LIN {X 0,Y 261.164,Z 765.318,A -85,B 0,C 180,E1 -18271.541,E2 -18271.541} C_VEL
LIN {X 0,Y 261.275,Z 764.733,A -85,B 0,C 180,E1 -18273.083,E2 -18273.083} C_VEL
LIN {X 0,Y 261.6,Z 762.413,A -85,B 0,C 180,E1 -18276.168,E2 -18276.168} C_VEL
LIN {X 0,Y 262.114,Z 759.545,A -85,B 0,C 180,E1 -18278.479,E2 -18278.479} C_VEL
LIN {X 0,Y 262.873,Z 755.654,A -85,B 0,C 180,E1 -18280.785,E2 -18280.785} C_VEL
LIN {X 0,Y 264.014,Z 750.637,A -85,B 0,C 180,E1 -18283.076,E2 -18283.076} C_VEL
LIN {X 0,Y 265.38,Z 744.319,A -85,B 0,C 180,E1 -18285.355,E2 -18285.355} C_VEL
LIN {X 0,Y 267.238,Z 736.403,A -85,B 0,C 180,E1 -18287.602,E2 -18287.602} C_VEL
LIN {X 0,Y 269.047,Z 728.334,A -85,B 0,C 180,E1 -18289.453,E2 -18289.453} C_VEL
LIN {X 0,Y 270.833,Z 718.491,A -85,B 0,C 180,E1 -18291.301,E2 -18291.301} C_VEL
LIN {X 0,Y 272.766,Z 707.41,A -85,B 0,C 180,E1 -18292.935,E2 -18292.935} C_VEL
LIN {X 0,Y 274.518,Z 696.535,A -85,B 0,C 180,E1 -18294.179,E2 -18294.179} C_VEL
LIN {X 0,Y 276.016,Z 684.51,A -85,B 0,C 180,E1 -18295.244,E2 -18295.244} C_VEL
LIN {X 0,Y 277.119,Z 672.156,A -85,B 0,C 180,E1 -18296.042,E2 -18296.042} C_VEL
LIN {X 0,Y 277.985,Z 659.336,A -85,B 0,C 180,E1 -18296.561,E2 -18296.561} C_VEL
LIN {X 0,Y 279.969,Z 592.257,A -85,B 0,C 180,E1 -18298.275,E2 -18298.275} C_VEL
LIN {X 0,Y 275.053,Z 579.197,A -85,B 0,C 180,E1 -18299.214,E2 -18299.214} C_VEL
LIN {X 0,Y 268.244,Z 564.095,A -85,B 0,C 180,E1 -18300.496,E2 -18300.496} C_VEL
LIN {X 0,Y 264.092,Z 555.532,A -85,B 0,C 180,E1 -18301.342,E2 -18301.342} C_VEL
LIN {X 0,Y 263.496,Z 553.165,A -85,B 0,C 180,E1 -18302.237,E2 -18302.237} C_VEL
LIN {X 0,Y 263.17,Z 551.724,A -85,B 0,C 180,E1 -18303.019,E2 -18303.019} C_VEL
LIN {X 0,Y 263.201,Z 551.693,A -85,B 0,C 180,E1 -18306.768,E2 -18306.768} C_VEL
LIN {X 0,Y 263.111,Z 551.696,A -85,B 0,C 180,E1 -18309.869,E2 -18309.869} C_VEL
LIN {X 0,Y 263.119,Z 551.693,A -85,B 0,C 180,E1 -18313.983,E2 -18313.983} C_VEL
LIN {X 0,Y 263.143,Z 551.706,A -85,B 0,C 180,E1 -18318.399,E2 -18318.399} C_VEL
LIN {X 0,Y 263.183,Z 551.673,A -85,B 0,C 180,E1 -18322.107,E2 -18322.107} C_VEL
LIN {X 0,Y 263.178,Z 551.702,A -85,B 0,C 180,E1 -18325.889,E2 -18325.889} C_VEL
LIN {X 0,Y 263.135,Z 551.7,A -85,B 0,C 180,E1 -18330.626,E2 -18330.626} C_VEL
LIN {X 0,Y 262.506,Z 551.779,A -85,B 0,C 180,E1 -18331.905,E2 -18331.905} C_VEL
LIN {X 0,Y 259.67,Z 552.137,A -85,B 0,C 180,E1 -18333.99,E2 -18333.99} C_VEL
LIN {X 0,Y 257.234,Z 552.441,A -85,B 0,C 180,E1 -18335.686,E2 -18335.686} C_VEL
LIN {X 0,Y 256.182,Z 552.564,A -85,B 0,C 180,E1 -18337.001,E2 -18337.001} C_VEL
LIN {X 0,Y 256.093,Z 552.571,A -85,B 0,C 180,E1 -18337.446,E2 -18337.446} C_VEL
LIN {X 0,Y 256.18,Z 552.572,A -85,B 0,C 180,E1 -18340.779,E2 -18340.779} C_VEL
LIN {X 0,Y 256.293,Z 552.544,A -85,B 0,C 180,E1 -18344.084,E2 -18344.084} C_VEL
LIN {X 0,Y 256.303,Z 552.548,A -85,B 0,C 180,E1 -18348.934,E2 -18348.934} C_VEL
LIN {X 0,Y 256.533,Z 552.526,A -85,B 0,C 180,E1 -18352.127,E2 -18352.127} C_VEL
LIN {X 0,Y 256.708,Z 552.501,A -85,B 0,C 180,E1 -18358.431,E2 -18358.431} C_VEL
LIN {X 0,Y 256.709,Z 552.503,A -85,B 0,C 180,E1 -18361.569,E2 -18361.569} C_VEL
LIN {X 0,Y 256.534,Z 552.526,A -85,B 0,C 180,E1 -18367.873,E2 -18367.873} C_VEL
LIN {X 0,Y 256.303,Z 552.545,A -85,B 0,C 180,E1 -18371.066,E2 -18371.066} C_VEL
LIN {X 0,Y 256.293,Z 552.545,A -85,B 0,C 180,E1 -18375.915,E2 -18375.915} C_VEL
LIN {X 0,Y 256.161,Z 552.568,A -85,B 0,C 180,E1 -18380.896,E2 -18380.896} C_VEL
LIN {X 0,Y 256.181,Z 552.573,A -85,B 0,C 180,E1 -18385.139,E2 -18385.139} C_VEL
LIN {X 0,Y 256.097,Z 552.584,A -85,B 0,C 180,E1 -18389.602,E2 -18389.602} C_VEL
LIN {X 0,Y 256.062,Z 552.59,A -85,B 0,C 180,E1 -18393.294,E2 -18393.294} C_VEL
LIN {X 0,Y 256.109,Z 552.557,A -85,B 0,C 180,E1 -18397.272,E2 -18397.272} C_VEL
LIN {X 0,Y 256.076,Z 552.575,A -85,B 0,C 180,E1 -18401.199,E2 -18401.199} C_VEL
LIN {X 0,Y 256.071,Z 552.585,A -85,B 0,C 180,E1 -18405.527,E2 -18405.527} C_VEL
LIN {X 0,Y 256.128,Z 552.582,A -85,B 0,C 180,E1 -18408.813,E2 -18408.813} C_VEL
LIN {X 0,Y 256.184,Z 552.737,A -85,B 0,C 180,E1 -18411.859,E2 -18411.859} C_VEL
LIN {X 0,Y 258.574,Z 562.726,A -85,B 0,C 180,E1 -18416.141,E2 -18416.141} C_VEL
LIN {X 0,Y 259.723,Z 567.866,A -85,B 0,C 180,E1 -18418.095,E2 -18418.095} C_VEL
LIN {X 0,Y 266.611,Z 583.7,A -85,B 0,C 180,E1 -18419.536,E2 -18419.536} C_VEL
LIN {X 0,Y 268.93,Z 589.726,A -85,B 0,C 180,E1 -18420.006,E2 -18420.006} C_VEL
LIN {X 0,Y 272.869,Z 615.019,A -85,B 0,C 180,E1 -18421.224,E2 -18421.224} C_VEL
LIN {X 0,Y 273.054,Z 619.058,A -85,B 0,C 180,E1 -18421.363,E2 -18421.363} C_VEL
LIN {X 0,Y 271.099,Z 676.352,A -85,B 0,C 180,E1 -18422.866,E2 -18422.866} C_VEL
LIN {X 0,Y 269.902,Z 690.247,A -85,B 0,C 180,E1 -18423.52,E2 -18423.52} C_VEL
LIN {X 0,Y 268.425,Z 702.691,A -85,B 0,C 180,E1 -18424.407,E2 -18424.407} C_VEL
LIN {X 0,Y 266.768,Z 713.801,A -85,B 0,C 180,E1 -18425.487,E2 -18425.487} C_VEL
LIN {X 0,Y 264.711,Z 725.369,A -85,B 0,C 180,E1 -18426.947,E2 -18426.947} C_VEL
LIN {X 0,Y 262.615,Z 735.787,A -85,B 0,C 180,E1 -18428.617,E2 -18428.617} C_VEL
LIN {X 0,Y 260.748,Z 744.664,A -85,B 0,C 180,E1 -18430.395,E2 -18430.395} C_VEL
LIN {X 0,Y 258.813,Z 753.554,A -85,B 0,C 180,E1 -18432.622,E2 -18432.622} C_VEL
LIN {X 0,Y 257.095,Z 760.984,A -85,B 0,C 180,E1 -18434.95,E2 -18434.95} C_VEL
LIN {X 0,Y 255.752,Z 766.951,A -85,B 0,C 180,E1 -18437.302,E2 -18437.302} C_VEL
LIN {X 0,Y 254.876,Z 771.673,A -85,B 0,C 180,E1 -18439.676,E2 -18439.676} C_VEL
LIN {X 0,Y 254.315,Z 775.286,A -85,B 0,C 180,E1 -18442.059,E2 -18442.059} C_VEL
LIN {X 0,Y 253.99,Z 778.347,A -85,B 0,C 180,E1 -18444.963,E2 -18444.963} C_VEL
LIN {X 0,Y 253.962,Z 779.544,A -85,B 0,C 180,E1 -18446.829,E2 -18446.829} C_VEL
LIN {X 0,Y 253.99,Z 780.152,A -85,B 0,C 180,E1 -18448.416,E2 -18448.416} C_VEL
LIN {X 0,Y 254.004,Z 780.51,A -85,B 0,C 180,E1 -18450.794,E2 -18450.794} C_VEL
LIN {X 0,Y 254.023,Z 782.645,A -85,B 0,C 180,E1 -18453.173,E2 -18453.173} C_VEL
LIN {X 0,Y 254.202,Z 783.607,A -85,B 0,C 180,E1 -18455.553,E2 -18455.553} C_VEL
LIN {X 0,Y 254.598,Z 783.41,A -85,B 0,C 180,E1 -18457.935,E2 -18457.935} C_VEL
LIN {X 0,Y 255.15,Z 782.591,A -85,B 0,C 180,E1 -18459.514,E2 -18459.514} C_VEL
LIN {X 0,Y 255.882,Z 781.29,A -85,B 0,C 180,E1 -18461.086,E2 -18461.086} C_VEL
LIN {X 0,Y 257.217,Z 778.306,A -85,B 0,C 180,E1 -18463.431,E2 -18463.431} C_VEL
LIN {X 0,Y 258.986,Z 774.096,A -85,B 0,C 180,E1 -18465.747,E2 -18465.747} C_VEL
LIN {X 0,Y 261.393,Z 768.401,A -85,B 0,C 180,E1 -18468.012,E2 -18468.012} C_VEL
LIN {X 0,Y 263.539,Z 762.327,A -85,B 0,C 180,E1 -18469.879,E2 -18469.879} C_VEL
LIN {X 0,Y 265.99,Z 754.985,A -85,B 0,C 180,E1 -18471.711,E2 -18471.711} C_VEL
LIN {X 0,Y 268.384,Z 746.866,A -85,B 0,C 180,E1 -18473.354,E2 -18473.354} C_VEL
LIN {X 0,Y 271.006,Z 736.903,A -85,B 0,C 180,E1 -18474.925,E2 -18474.925} C_VEL
LIN {X 0,Y 273.235,Z 727.291,A -85,B 0,C 180,E1 -18476.136,E2 -18476.136} C_VEL
LIN {X 0,Y 275.407,Z 716.047,A -85,B 0,C 180,E1 -18477.243,E2 -18477.243} C_VEL
LIN {X 0,Y 277.242,Z 703.03,A -85,B 0,C 180,E1 -18478.174,E2 -18478.174} C_VEL
LIN {X 0,Y 280.075,Z 679.812,A -85,B 0,C 180,E1 -18479.4,E2 -18479.4} C_VEL
LIN {X 0,Y 288.139,Z 623.235,A -85,B 0,C 180,E1 -18482.092,E2 -18482.092} C_VEL
LIN {X 0,Y 288.371,Z 616.794,A -85,B 0,C 180,E1 -18482.75,E2 -18482.75} C_VEL
LIN {X 0,Y 288.876,Z 615.038,A -85,B 0,C 180,E1 -18483.011,E2 -18483.011} C_VEL
LIN {X 0,Y 289.022,Z 612.57,A -85,B 0,C 180,E1 -18483.645,E2 -18483.645} C_VEL
LIN {X 0,Y 288.692,Z 608.855,A -85,B 0,C 180,E1 -18484.984,E2 -18484.984} C_VEL
LIN {X 0,Y 287.679,Z 606.935,A -85,B 0,C 180,E1 -18486.274,E2 -18486.274} C_VEL
LIN {X 0,Y 286.249,Z 605.014,A -85,B 0,C 180,E1 -18488.218,E2 -18488.218} C_VEL
LIN {X 0,Y 285.184,Z 603.787,A -85,B 0,C 180,E1 -18490.186,E2 -18490.186} C_VEL
LIN {X 0,Y 284.41,Z 603.27,A -85,B 0,C 180,E1 -18492.156,E2 -18492.156} C_VEL
LIN {X 0,Y 283.942,Z 603.412,A -85,B 0,C 180,E1 -18494.127,E2 -18494.127} C_VEL
LIN {X 0,Y 283.705,Z 604.229,A -85,B 0,C 180,E1 -18496.082,E2 -18496.082} C_VEL
LIN {X 0,Y 283.644,Z 606.871,A -85,B 0,C 180,E1 -18499.151,E2 -18499.151} C_VEL
LIN {X 0,Y 283.702,Z 608.841,A -85,B 0,C 180,E1 -18500.696,E2 -18500.696} C_VEL
LIN {X 0,Y 283.768,Z 613.689,A -85,B 0,C 180,E1 -18503.53,E2 -18503.53} C_VEL
LIN {X 0,Y 283.557,Z 617.891,A -85,B 0,C 180,E1 -18505.354,E2 -18505.354} C_VEL
LIN {X 0,Y 284.753,Z 629.469,A -85,B 0,C 180,E1 -18507.242,E2 -18507.242} C_VEL
LIN {X 0,Y 286.092,Z 642.547,A -85,B 0,C 180,E1 -18509.032,E2 -18509.032} C_VEL
LIN {X 0,Y 286.986,Z 654.978,A -85,B 0,C 180,E1 -18510.424,E2 -18510.424} C_VEL
LIN {X 0,Y 287.008,Z 657.879,A -85,B 0,C 180,E1 -18510.676,E2 -18510.676} C_VEL
LIN {X 0,Y 281.094,Z 703.082,A -85,B 0,C 180,E1 -18512.802,E2 -18512.802} C_VEL
LIN {X 0,Y 278.886,Z 715.353,A -85,B 0,C 180,E1 -18513.631,E2 -18513.631} C_VEL
LIN {X 0,Y 276.564,Z 725.576,A -85,B 0,C 180,E1 -18514.607,E2 -18514.607} C_VEL
LIN {X 0,Y 273.969,Z 735.191,A -85,B 0,C 180,E1 -18515.767,E2 -18515.767} C_VEL
LIN {X 0,Y 271.23,Z 744.198,A -85,B 0,C 180,E1 -18517.128,E2 -18517.128} C_VEL
LIN {X 0,Y 268.708,Z 751.51,A -85,B 0,C 180,E1 -18518.521,E2 -18518.521} C_VEL
LIN {X 0,Y 266.368,Z 757.638,A -85,B 0,C 180,E1 -18519.94,E2 -18519.94} C_VEL
LIN {X 0,Y 263.79,Z 763.91,A -85,B 0,C 180,E1 -18521.757,E2 -18521.757} C_VEL
LIN {X 0,Y 261.577,Z 769.036,A -85,B 0,C 180,E1 -18523.614,E2 -18523.614} C_VEL
LIN {X 0,Y 259.179,Z 773.831,A -85,B 0,C 180,E1 -18525.874,E2 -18525.874} C_VEL
LIN {X 0,Y 257.853,Z 776.163,A -85,B 0,C 180,E1 -18527.406,E2 -18527.406} C_VEL
LIN {X 0,Y 256.787,Z 777.941,A -85,B 0,C 180,E1 -18528.955,E2 -18528.955} C_VEL
LIN {X 0,Y 255.908,Z 779.221,A -85,B 0,C 180,E1 -18530.516,E2 -18530.516} C_VEL
LIN {X 0,Y 254.98,Z 780.156,A -85,B 0,C 180,E1 -18532.876,E2 -18532.876} C_VEL
LIN {X 0,Y 254.312,Z 779.949,A -85,B 0,C 180,E1 -18535.244,E2 -18535.244} C_VEL
LIN {X 0,Y 254.099,Z 779.107,A -85,B 0,C 180,E1 -18536.829,E2 -18536.829} C_VEL
LIN {X 0,Y 254.042,Z 777.756,A -85,B 0,C 180,E1 -18538.415,E2 -18538.415} C_VEL
LIN {X 0,Y 253.998,Z 774.661,A -85,B 0,C 180,E1 -18540.793,E2 -18540.793} C_VEL
LIN {X 0,Y 254.205,Z 770.236,A -85,B 0,C 180,E1 -18543.17,E2 -18543.17} C_VEL
LIN {X 0,Y 254.33,Z 765.193,A -85,B 0,C 180,E1 -18545.165,E2 -18545.165} C_VEL
LIN {X 0,Y 254.692,Z 758.914,A -85,B 0,C 180,E1 -18547.133,E2 -18547.133} C_VEL
LIN {X 0,Y 254.949,Z 752.669,A -85,B 0,C 180,E1 -18548.721,E2 -18548.721} C_VEL
LIN {X 0,Y 255.484,Z 744.165,A -85,B 0,C 180,E1 -18550.501,E2 -18550.501} C_VEL
LIN {X 0,Y 256.12,Z 734.618,A -85,B 0,C 180,E1 -18552.077,E2 -18552.077} C_VEL
LIN {X 0,Y 256.642,Z 725.68,A -85,B 0,C 180,E1 -18553.259,E2 -18553.259} C_VEL
LIN {X 0,Y 257.255,Z 714.434,A -85,B 0,C 180,E1 -18554.436,E2 -18554.436} C_VEL
LIN {X 0,Y 257.657,Z 702.446,A -85,B 0,C 180,E1 -18555.322,E2 -18555.322} C_VEL
LIN {X 0,Y 258.25,Z 687.986,A -85,B 0,C 180,E1 -18556.045,E2 -18556.045} C_VEL
LIN {X 0,Y 259.335,Z 642.712,A -85,B 0,C 180,E1 -18558.044,E2 -18558.044} C_VEL
LIN {X 0,Y 257.654,Z 620.795,A -85,B 0,C 180,E1 -18559.034,E2 -18559.034} C_VEL
LIN {X 0,Y 257.61,Z 617.12,A -85,B 0,C 180,E1 -18559.265,E2 -18559.265} C_VEL
LIN {X 0,Y 259.319,Z 596.268,A -85,B 0,C 180,E1 -18563.987,E2 -18563.987} C_VEL
LIN {X 0,Y 261.02,Z 578.045,A -85,B 0,C 180,E1 -18568.112,E2 -18568.112} C_VEL
LIN {X 0,Y 260.619,Z 574.104,A -85,B 0,C 180,E1 -18569.039,E2 -18569.039} C_VEL
LIN {X 0,Y 256.597,Z 554.39,A -85,B 0,C 180,E1 -18573.892,E2 -18573.892} C_VEL
LIN {X 0,Y 256.23,Z 552.679,A -85,B 0,C 180,E1 -18574.402,E2 -18574.402} C_VEL
LIN {X 0,Y 256.133,Z 552.582,A -85,B 0,C 180,E1 -18577.275,E2 -18577.275} C_VEL
LIN {X 0,Y 256.06,Z 552.532,A -85,B 0,C 180,E1 -18581.203,E2 -18581.203} C_VEL
LIN {X 0,Y 256.058,Z 552.579,A -85,B 0,C 180,E1 -18585.53,E2 -18585.53} C_VEL
LIN {X 0,Y 256.058,Z 552.558,A -85,B 0,C 180,E1 -18588.796,E2 -18588.796} C_VEL
LIN {X 0,Y 256.134,Z 552.57,A -85,B 0,C 180,E1 -18592.867,E2 -18592.867} C_VEL
LIN {X 0,Y 256.153,Z 552.695,A -85,B 0,C 180,E1 -18596.5,E2 -18596.5} C_VEL
LIN {X 0,Y 256.89,Z 555.635,A -85,B 0,C 180,E1 -18597.795,E2 -18597.795} C_VEL
LIN {X 0,Y 264.902,Z 572.152,A -85,B 0,C 180,E1 -18599.454,E2 -18599.454} C_VEL
LIN {X 0,Y 271.815,Z 588.544,A -85,B 0,C 180,E1 -18600.806,E2 -18600.806} C_VEL
LIN {X 0,Y 273.595,Z 593.413,A -85,B 0,C 180,E1 -18601.159,E2 -18601.159} C_VEL
LIN {X 0,Y 271.464,Z 661.742,A -85,B 0,C 180,E1 -18602.955,E2 -18602.955} C_VEL
LIN {X 0,Y 270.465,Z 675.096,A -85,B 0,C 180,E1 -18603.576,E2 -18603.576} C_VEL
LIN {X 0,Y 269.157,Z 687.837,A -85,B 0,C 180,E1 -18604.478,E2 -18604.478} C_VEL
LIN {X 0,Y 267.605,Z 699.142,A -85,B 0,C 180,E1 -18605.565,E2 -18605.565} C_VEL
LIN {X 0,Y 265.672,Z 710.779,A -85,B 0,C 180,E1 -18607.032,E2 -18607.032} C_VEL
LIN {X 0,Y 263.921,Z 719.999,A -85,B 0,C 180,E1 -18608.489,E2 -18608.489} C_VEL
LIN {X 0,Y 262.068,Z 729.758,A -85,B 0,C 180,E1 -18610.413,E2 -18610.413} C_VEL
LIN {X 0,Y 260.246,Z 737.623,A -85,B 0,C 180,E1 -18612.312,E2 -18612.312} C_VEL
LIN {X 0,Y 258.368,Z 745.306,A -85,B 0,C 180,E1 -18614.619,E2 -18614.619} C_VEL
LIN {X 0,Y 256.723,Z 752.357,A -85,B 0,C 180,E1 -18617.348,E2 -18617.348} C_VEL
LIN {X 0,Y 255.59,Z 757.052,A -85,B 0,C 180,E1 -18619.703,E2 -18619.703} C_VEL
LIN {X 0,Y 254.885,Z 760.637,A -85,B 0,C 180,E1 -18622.074,E2 -18622.074} C_VEL
LIN {X 0,Y 254.515,Z 762.598,A -85,B 0,C 180,E1 -18623.765,E2 -18623.765} C_VEL
LIN {X 0,Y 254.194,Z 764.873,A -85,B 0,C 180,E1 -18626.829,E2 -18626.829} C_VEL
LIN {X 0,Y 254.096,Z 765.484,A -85,B 0,C 180,E1 -18628.414,E2 -18628.414} C_VEL
LIN {X 0,Y 254.064,Z 765.714,A -85,B 0,C 180,E1 -18629.999,E2 -18629.999} C_VEL
LIN {X 0,Y 254.095,Z 765.522,A -85,B 0,C 180,E1 -18631.584,E2 -18631.584} C_VEL
LIN {X 0,Y 254.192,Z 764.937,A -85,B 0,C 180,E1 -18633.169,E2 -18633.169} C_VEL
LIN {X 0,Y 254.534,Z 762.617,A -85,B 0,C 180,E1 -18636.34,E2 -18636.34} C_VEL
LIN {X 0,Y 255.077,Z 759.749,A -85,B 0,C 180,E1 -18638.715,E2 -18638.715} C_VEL
LIN {X 0,Y 255.91,Z 755.858,A -85,B 0,C 180,E1 -18641.082,E2 -18641.082} C_VEL
LIN {X 0,Y 257.1,Z 750.84,A -85,B 0,C 180,E1 -18643.434,E2 -18643.434} C_VEL
LIN {X 0,Y 258.531,Z 744.522,A -85,B 0,C 180,E1 -18645.772,E2 -18645.772} C_VEL
LIN {X 0,Y 260.488,Z 736.605,A -85,B 0,C 180,E1 -18648.074,E2 -18648.074} C_VEL
LIN {X 0,Y 262.351,Z 728.536,A -85,B 0,C 180,E1 -18649.97,E2 -18649.97} C_VEL
LIN {X 0,Y 264.24,Z 718.692,A -85,B 0,C 180,E1 -18651.86,E2 -18651.86} C_VEL
LIN {X 0,Y 266.263,Z 707.609,A -85,B 0,C 180,E1 -18653.528,E2 -18653.528} C_VEL
LIN {X 0,Y 268.081,Z 696.733,A -85,B 0,C 180,E1 -18654.799,E2 -18654.799} C_VEL
LIN {X 0,Y 269.634,Z 684.707,A -85,B 0,C 180,E1 -18655.885,E2 -18655.885} C_VEL
LIN {X 0,Y 270.773,Z 672.349,A -85,B 0,C 180,E1 -18656.7,E2 -18656.7} C_VEL
LIN {X 0,Y 271.674,Z 659.519,A -85,B 0,C 180,E1 -18657.228,E2 -18657.228} C_VEL
LIN {X 0,Y 273.728,Z 593.61,A -85,B 0,C 180,E1 -18658.946,E2 -18658.946} C_VEL
LIN {X 0,Y 266.65,Z 575.931,A -85,B 0,C 180,E1 -18660.336,E2 -18660.336} C_VEL
LIN {X 0,Y 258.475,Z 558.972,A -85,B 0,C 180,E1 -18661.954,E2 -18661.954} C_VEL
LIN {X 0,Y 256.796,Z 555.428,A -85,B 0,C 180,E1 -18662.39,E2 -18662.39} C_VEL
LIN {X 0,Y 256.138,Z 552.622,A -85,B 0,C 180,E1 -18663.719,E2 -18663.719} C_VEL
LIN {X 0,Y 256.127,Z 552.578,A -85,B 0,C 180,E1 -18667.274,E2 -18667.274} C_VEL
LIN {X 0,Y 256.053,Z 552.584,A -85,B 0,C 180,E1 -18671.201,E2 -18671.201} C_VEL
LIN {X 0,Y 256.057,Z 552.569,A -85,B 0,C 180,E1 -18675.528,E2 -18675.528} C_VEL
LIN {X 0,Y 256.079,Z 552.582,A -85,B 0,C 180,E1 -18678.801,E2 -18678.801} C_VEL
LIN {X 0,Y 256.149,Z 552.557,A -85,B 0,C 180,E1 -18682.87,E2 -18682.87} C_VEL
LIN {X 0,Y 256.08,Z 552.582,A -85,B 0,C 180,E1 -18686.709,E2 -18686.709} C_VEL
LIN {X 0,Y 256.133,Z 552.572,A -85,B 0,C 180,E1 -18691.404,E2 -18691.404} C_VEL
LIN {X 0,Y 256.161,Z 552.574,A -85,B 0,C 180,E1 -18695.698,E2 -18695.698} C_VEL
LIN {X 0,Y 256.093,Z 552.571,A -85,B 0,C 180,E1 -18697.446,E2 -18697.446} C_VEL
LIN {X 0,Y 255.437,Z 552.656,A -85,B 0,C 180,E1 -18698.76,E2 -18698.76} C_VEL
LIN {X 0,Y 252.66,Z 553.011,A -85,B 0,C 180,E1 -18700.904,E2 -18700.904} C_VEL
LIN {X 0,Y 250.299,Z 553.296,A -85,B 0,C 180,E1 -18702.649,E2 -18702.649} C_VEL
LIN {X 0,Y 249.279,Z 553.417,A -85,B 0,C 180,E1 -18704,E2 -18704} C_VEL
LIN {X 0,Y 249.191,Z 553.428,A -85,B 0,C 180,E1 -18704.457,E2 -18704.457} C_VEL
LIN {X 0,Y 249.246,Z 553.43,A -85,B 0,C 180,E1 -18708.616,E2 -18708.616} C_VEL
LIN {X 0,Y 249.475,Z 553.401,A -85,B 0,C 180,E1 -18711.903,E2 -18711.903} C_VEL
LIN {X 0,Y 249.43,Z 553.396,A -85,B 0,C 180,E1 -18716.769,E2 -18716.769} C_VEL
LIN {X 0,Y 249.729,Z 553.378,A -85,B 0,C 180,E1 -18720,E2 -18720} C_VEL
LIN {X 0,Y 249.431,Z 553.398,A -85,B 0,C 180,E1 -18723.23,E2 -18723.23} C_VEL
LIN {X 0,Y 249.478,Z 553.404,A -85,B 0,C 180,E1 -18728.097,E2 -18728.097} C_VEL
LIN {X 0,Y 249.247,Z 553.426,A -85,B 0,C 180,E1 -18731.384,E2 -18731.384} C_VEL
LIN {X 0,Y 249.235,Z 553.424,A -85,B 0,C 180,E1 -18736.379,E2 -18736.379} C_VEL
LIN {X 0,Y 249.081,Z 553.447,A -85,B 0,C 180,E1 -18741.519,E2 -18741.519} C_VEL
LIN {X 0,Y 249.124,Z 553.448,A -85,B 0,C 180,E1 -18745.482,E2 -18745.482} C_VEL
LIN {X 0,Y 249.066,Z 553.461,A -85,B 0,C 180,E1 -18748.99,E2 -18748.99} C_VEL
LIN {X 0,Y 249.025,Z 553.465,A -85,B 0,C 180,E1 -18752.427,E2 -18752.427} C_VEL
LIN {X 0,Y 249.024,Z 553.436,A -85,B 0,C 180,E1 -18756.346,E2 -18756.346} C_VEL
LIN {X 0,Y 249.03,Z 553.464,A -85,B 0,C 180,E1 -18760.473,E2 -18760.473} C_VEL
LIN {X 0,Y 249.015,Z 553.468,A -85,B 0,C 180,E1 -18764.876,E2 -18764.876} C_VEL
LIN {X 0,Y 249.077,Z 553.446,A -85,B 0,C 180,E1 -18767.378,E2 -18767.378} C_VEL
LIN {X 0,Y 249.119,Z 553.651,A -85,B 0,C 180,E1 -18771.056,E2 -18771.056} C_VEL
LIN {X 0,Y 250.889,Z 560.889,A -85,B 0,C 180,E1 -18774.327,E2 -18774.327} C_VEL
LIN {X 0,Y 252.416,Z 567.595,A -85,B 0,C 180,E1 -18777.053,E2 -18777.053} C_VEL
LIN {X 0,Y 259.177,Z 582.558,A -85,B 0,C 180,E1 -18778.535,E2 -18778.535} C_VEL
LIN {X 0,Y 263.074,Z 592.539,A -85,B 0,C 180,E1 -18779.36,E2 -18779.36} C_VEL
LIN {X 0,Y 266.842,Z 617.494,A -85,B 0,C 180,E1 -18780.591,E2 -18780.591} C_VEL
LIN {X 0,Y 264.803,Z 676.161,A -85,B 0,C 180,E1 -18782.165,E2 -18782.165} C_VEL
LIN {X 0,Y 263.58,Z 690.052,A -85,B 0,C 180,E1 -18782.833,E2 -18782.833} C_VEL
LIN {X 0,Y 262.025,Z 702.492,A -85,B 0,C 180,E1 -18783.734,E2 -18783.734} C_VEL
LIN {X 0,Y 260.31,Z 713.601,A -85,B 0,C 180,E1 -18784.837,E2 -18784.837} C_VEL
LIN {X 0,Y 258.165,Z 725.167,A -85,B 0,C 180,E1 -18786.327,E2 -18786.327} C_VEL
LIN {X 0,Y 255.999,Z 735.585,A -85,B 0,C 180,E1 -18788.036,E2 -18788.036} C_VEL
LIN {X 0,Y 254.118,Z 744.109,A -85,B 0,C 180,E1 -18789.777,E2 -18789.777} C_VEL
LIN {X 0,Y 252.363,Z 752.158,A -85,B 0,C 180,E1 -18791.797,E2 -18791.797} C_VEL
LIN {X 0,Y 250.528,Z 759.66,A -85,B 0,C 180,E1 -18794.128,E2 -18794.128} C_VEL
LIN {X 0,Y 248.79,Z 766.747,A -85,B 0,C 180,E1 -18796.94,E2 -18796.94} C_VEL
LIN {X 0,Y 247.858,Z 771.468,A -85,B 0,C 180,E1 -18799.381,E2 -18799.381} C_VEL
LIN {X 0,Y 247.267,Z 775.082,A -85,B 0,C 180,E1 -18801.831,E2 -18801.831} C_VEL
LIN {X 0,Y 247.009,Z 776.944,A -85,B 0,C 180,E1 -18803.466,E2 -18803.466} C_VEL
LIN {X 0,Y 246.882,Z 778.341,A -85,B 0,C 180,E1 -18805.102,E2 -18805.102} C_VEL
LIN {X 0,Y 246.865,Z 779.339,A -85,B 0,C 180,E1 -18806.737,E2 -18806.737} C_VEL
LIN {X 0,Y 246.9,Z 779.948,A -85,B 0,C 180,E1 -18808.37,E2 -18808.37} C_VEL
LIN {X 0,Y 246.939,Z 780.108,A -85,B 0,C 180,E1 -18811.021,E2 -18811.021} C_VEL
LIN {X 0,Y 246.945,Z 782.262,A -85,B 0,C 180,E1 -18813.264,E2 -18813.264} C_VEL
LIN {X 0,Y 247.089,Z 783.383,A -85,B 0,C 180,E1 -18815.429,E2 -18815.429} C_VEL
LIN {X 0,Y 247.563,Z 783.464,A -85,B 0,C 180,E1 -18818.162,E2 -18818.162} C_VEL
LIN {X 0,Y 248.162,Z 782.873,A -85,B 0,C 180,E1 -18819.785,E2 -18819.785} C_VEL
LIN {X 0,Y 248.944,Z 781.787,A -85,B 0,C 180,E1 -18821.399,E2 -18821.399} C_VEL
LIN {X 0,Y 250.355,Z 779.09,A -85,B 0,C 180,E1 -18823.806,E2 -18823.806} C_VEL
LIN {X 0,Y 252.25,Z 775.164,A -85,B 0,C 180,E1 -18826.179,E2 -18826.179} C_VEL
LIN {X 0,Y 254.791,Z 769.872,A -85,B 0,C 180,E1 -18828.496,E2 -18828.496} C_VEL
LIN {X 0,Y 257.614,Z 763.042,A -85,B 0,C 180,E1 -18830.774,E2 -18830.774} C_VEL
LIN {X 0,Y 260.063,Z 756.333,A -85,B 0,C 180,E1 -18832.517,E2 -18832.517} C_VEL
LIN {X 0,Y 262.392,Z 749.327,A -85,B 0,C 180,E1 -18834.036,E2 -18834.036} C_VEL
LIN {X 0,Y 265.402,Z 739.699,A -85,B 0,C 180,E1 -18835.699,E2 -18835.699} C_VEL
LIN {X 0,Y 268.119,Z 729.217,A -85,B 0,C 180,E1 -18837.094,E2 -18837.094} C_VEL
LIN {X 0,Y 270.291,Z 719.596,A -85,B 0,C 180,E1 -18838.119,E2 -18838.119} C_VEL
LIN {X 0,Y 272.514,Z 707.097,A -85,B 0,C 180,E1 -18839.13,E2 -18839.13} C_VEL
LIN {X 0,Y 274.79,Z 689.707,A -85,B 0,C 180,E1 -18840.129,E2 -18840.129} C_VEL
LIN {X 0,Y 284.58,Z 625.063,A -85,B 0,C 180,E1 -18843.284,E2 -18843.284} C_VEL
LIN {X 0,Y 284.762,Z 618.517,A -85,B 0,C 180,E1 -18843.946,E2 -18843.946} C_VEL
LIN {X 0,Y 284.547,Z 616.843,A -85,B 0,C 180,E1 -18844.365,E2 -18844.365} C_VEL
LIN {X 0,Y 284.339,Z 614.215,A -85,B 0,C 180,E1 -18845.347,E2 -18845.347} C_VEL
LIN {X 0,Y 282.791,Z 611.68,A -85,B 0,C 180,E1 -18847.319,E2 -18847.319} C_VEL
LIN {X 0,Y 281.504,Z 610.085,A -85,B 0,C 180,E1 -18849.29,E2 -18849.29} C_VEL
LIN {X 0,Y 280.517,Z 609.207,A -85,B 0,C 180,E1 -18851.27,E2 -18851.27} C_VEL
LIN {X 0,Y 279.851,Z 609.01,A -85,B 0,C 180,E1 -18853.257,E2 -18853.257} C_VEL
LIN {X 0,Y 279.407,Z 609.494,A -85,B 0,C 180,E1 -18855.228,E2 -18855.228} C_VEL
LIN {X 0,Y 279.15,Z 610.667,A -85,B 0,C 180,E1 -18857.175,E2 -18857.175} C_VEL
LIN {X 0,Y 279.082,Z 613.325,A -85,B 0,C 180,E1 -18859.915,E2 -18859.915} C_VEL
LIN {X 0,Y 278.948,Z 617.866,A -85,B 0,C 180,E1 -18862.795,E2 -18862.795} C_VEL
LIN {X 0,Y 280.508,Z 623.055,A -85,B 0,C 180,E1 -18864.563,E2 -18864.563} C_VEL
LIN {X 0,Y 281.613,Z 636.846,A -85,B 0,C 180,E1 -18866.787,E2 -18866.787} C_VEL
LIN {X 0,Y 282.492,Z 649.442,A -85,B 0,C 180,E1 -18868.473,E2 -18868.473} C_VEL
LIN {X 0,Y 282.893,Z 659.147,A -85,B 0,C 180,E1 -18869.542,E2 -18869.542} C_VEL
LIN {X 0,Y 276.762,Z 702.685,A -85,B 0,C 180,E1 -18871.619,E2 -18871.619} C_VEL
LIN {X 0,Y 274.619,Z 713.885,A -85,B 0,C 180,E1 -18872.364,E2 -18872.364} C_VEL
LIN {X 0,Y 271.734,Z 725.886,A -85,B 0,C 180,E1 -18873.503,E2 -18873.503} C_VEL
LIN {X 0,Y 268.986,Z 735.508,A -85,B 0,C 180,E1 -18874.669,E2 -18874.669} C_VEL
LIN {X 0,Y 265.709,Z 745.328,A -85,B 0,C 180,E1 -18876.211,E2 -18876.211} C_VEL
LIN {X 0,Y 262.994,Z 752.402,A -85,B 0,C 180,E1 -18877.617,E2 -18877.617} C_VEL
LIN {X 0,Y 259.943,Z 759.741,A -85,B 0,C 180,E1 -18879.422,E2 -18879.422} C_VEL
LIN {X 0,Y 256.743,Z 766.755,A -85,B 0,C 180,E1 -18881.651,E2 -18881.651} C_VEL
LIN {X 0,Y 254.046,Z 771.968,A -85,B 0,C 180,E1 -18883.94,E2 -18883.94} C_VEL
LIN {X 0,Y 251.687,Z 775.909,A -85,B 0,C 180,E1 -18886.27,E2 -18886.27} C_VEL
LIN {X 0,Y 249.871,Z 778.588,A -85,B 0,C 180,E1 -18888.645,E2 -18888.645} C_VEL
LIN {X 0,Y 248.925,Z 779.623,A -85,B 0,C 180,E1 -18890.247,E2 -18890.247} C_VEL
LIN {X 0,Y 247.793,Z 780.343,A -85,B 0,C 180,E1 -18893.072,E2 -18893.072} C_VEL
LIN {X 0,Y 247.244,Z 779.845,A -85,B 0,C 180,E1 -18895.108,E2 -18895.108} C_VEL
LIN {X 0,Y 247.026,Z 778.84,A -85,B 0,C 180,E1 -18896.738,E2 -18896.738} C_VEL
LIN {X 0,Y 246.933,Z 776.379,A -85,B 0,C 180,E1 -18899.185,E2 -18899.185} C_VEL
LIN {X 0,Y 246.984,Z 772.505,A -85,B 0,C 180,E1 -18901.631,E2 -18901.631} C_VEL
LIN {X 0,Y 247.232,Z 767.192,A -85,B 0,C 180,E1 -18904.075,E2 -18904.075} C_VEL
LIN {X 0,Y 247.541,Z 760.096,A -85,B 0,C 180,E1 -18906.521,E2 -18906.521} C_VEL
LIN {X 0,Y 247.807,Z 754.111,A -85,B 0,C 180,E1 -18908.152,E2 -18908.152} C_VEL
LIN {X 0,Y 248.213,Z 746.906,A -85,B 0,C 180,E1 -18909.781,E2 -18909.781} C_VEL
LIN {X 0,Y 248.789,Z 738.186,A -85,B 0,C 180,E1 -18911.405,E2 -18911.405} C_VEL
LIN {X 0,Y 249.484,Z 727.082,A -85,B 0,C 180,E1 -18913.024,E2 -18913.024} C_VEL
LIN {X 0,Y 250.05,Z 717.155,A -85,B 0,C 180,E1 -18914.133,E2 -18914.133} C_VEL
LIN {X 0,Y 250.468,Z 705.188,A -85,B 0,C 180,E1 -18915.148,E2 -18915.148} C_VEL
LIN {X 0,Y 251.02,Z 691.705,A -85,B 0,C 180,E1 -18915.894,E2 -18915.894} C_VEL
LIN {X 0,Y 252.307,Z 643.671,A -85,B 0,C 180,E1 -18918.093,E2 -18918.093} C_VEL
LIN {X 0,Y 250.581,Z 620.824,A -85,B 0,C 180,E1 -18919.177,E2 -18919.177} C_VEL
LIN {X 0,Y 250.551,Z 617.295,A -85,B 0,C 180,E1 -18919.376,E2 -18919.376} C_VEL
LIN {X 0,Y 252.323,Z 596.175,A -85,B 0,C 180,E1 -18924.257,E2 -18924.257} C_VEL
LIN {X 0,Y 253.95,Z 579.679,A -85,B 0,C 180,E1 -18928.065,E2 -18928.065} C_VEL
LIN {X 0,Y 253.715,Z 575.774,A -85,B 0,C 180,E1 -18928.997,E2 -18928.997} C_VEL
LIN {X 0,Y 249.762,Z 556.397,A -85,B 0,C 180,E1 -18933.84,E2 -18933.84} C_VEL
LIN {X 0,Y 249.174,Z 553.587,A -85,B 0,C 180,E1 -18934.626,E2 -18934.626} C_VEL
LIN {X 0,Y 249.043,Z 553.458,A -85,B 0,C 180,E1 -18938.378,E2 -18938.378} C_VEL
LIN {X 0,Y 249.005,Z 553.406,A -85,B 0,C 180,E1 -18942.79,E2 -18942.79} C_VEL
LIN {X 0,Y 249.02,Z 553.462,A -85,B 0,C 180,E1 -18947.362,E2 -18947.362} C_VEL
LIN {X 0,Y 249.047,Z 553.437,A -85,B 0,C 180,E1 -18952.2,E2 -18952.2} C_VEL
LIN {X 0,Y 249.068,Z 553.518,A -85,B 0,C 180,E1 -18955.642,E2 -18955.642} C_VEL
LIN {X 0,Y 249.562,Z 555.442,A -85,B 0,C 180,E1 -18956.621,E2 -18956.621} C_VEL
LIN {X 0,Y 250.068,Z 556.886,A -85,B 0,C 180,E1 -18956.882,E2 -18956.882} C_VEL
LIN {X 0,Y 257.618,Z 571.872,A -85,B 0,C 180,E1 -18958.475,E2 -18958.475} C_VEL
LIN {X 0,Y 263.259,Z 584.586,A -85,B 0,C 180,E1 -18959.627,E2 -18959.627} C_VEL
LIN {X 0,Y 267.424,Z 595.311,A -85,B 0,C 180,E1 -18960.479,E2 -18960.479} C_VEL
LIN {X 0,Y 265.18,Z 661.963,A -85,B 0,C 180,E1 -18962.259,E2 -18962.259} C_VEL
LIN {X 0,Y 264.132,Z 675.31,A -85,B 0,C 180,E1 -18962.891,E2 -18962.891} C_VEL
LIN {X 0,Y 262.783,Z 688.049,A -85,B 0,C 180,E1 -18963.813,E2 -18963.813} C_VEL
LIN {X 0,Y 261.179,Z 699.352,A -85,B 0,C 180,E1 -18964.923,E2 -18964.923} C_VEL
LIN {X 0,Y 259.16,Z 710.988,A -85,B 0,C 180,E1 -18966.421,E2 -18966.421} C_VEL
LIN {X 0,Y 257.077,Z 721.435,A -85,B 0,C 180,E1 -18968.129,E2 -18968.129} C_VEL
LIN {X 0,Y 255.393,Z 729.966,A -85,B 0,C 180,E1 -18969.879,E2 -18969.879} C_VEL
LIN {X 0,Y 253.491,Z 737.83,A -85,B 0,C 180,E1 -18971.825,E2 -18971.825} C_VEL
LIN {X 0,Y 251.504,Z 745.513,A -85,B 0,C 180,E1 -18974.188,E2 -18974.188} C_VEL
LIN {X 0,Y 250.256,Z 750.756,A -85,B 0,C 180,E1 -18976.188,E2 -18976.188} C_VEL
LIN {X 0,Y 248.951,Z 755.843,A -85,B 0,C 180,E1 -18978.601,E2 -18978.601} C_VEL
LIN {X 0,Y 248.068,Z 759.785,A -85,B 0,C 180,E1 -18981.034,E2 -18981.034} C_VEL
LIN {X 0,Y 247.424,Z 763.002,A -85,B 0,C 180,E1 -18983.81,E2 -18983.81} C_VEL
LIN {X 0,Y 247.114,Z 765.078,A -85,B 0,C 180,E1 -18986.738,E2 -18986.738} C_VEL
LIN {X 0,Y 246.993,Z 765.918,A -85,B 0,C 180,E1 -18989.999,E2 -18989.999} C_VEL
LIN {X 0,Y 247.006,Z 765.726,A -85,B 0,C 180,E1 -18991.629,E2 -18991.629} C_VEL
LIN {X 0,Y 247.111,Z 765.141,A -85,B 0,C 180,E1 -18993.259,E2 -18993.259} C_VEL
LIN {X 0,Y 247.495,Z 762.821,A -85,B 0,C 180,E1 -18996.521,E2 -18996.521} C_VEL
LIN {X 0,Y 248.066,Z 759.953,A -85,B 0,C 180,E1 -18998.963,E2 -18998.963} C_VEL
LIN {X 0,Y 248.929,Z 756.062,A -85,B 0,C 180,E1 -19001.397,E2 -19001.397} C_VEL
LIN {X 0,Y 250.184,Z 751.044,A -85,B 0,C 180,E1 -19003.813,E2 -19003.813} C_VEL
LIN {X 0,Y 251.703,Z 744.724,A -85,B 0,C 180,E1 -19006.212,E2 -19006.212} C_VEL
LIN {X 0,Y 253.758,Z 736.807,A -85,B 0,C 180,E1 -19008.571,E2 -19008.571} C_VEL
LIN {X 0,Y 255.68,Z 728.738,A -85,B 0,C 180,E1 -19010.514,E2 -19010.514} C_VEL
LIN {X 0,Y 257.652,Z 718.894,A -85,B 0,C 180,E1 -19012.449,E2 -19012.449} C_VEL
LIN {X 0,Y 259.787,Z 707.809,A -85,B 0,C 180,E1 -19014.151,E2 -19014.151} C_VEL
LIN {X 0,Y 261.666,Z 696.931,A -85,B 0,C 180,E1 -19015.449,E2 -19015.449} C_VEL
LIN {X 0,Y 263.266,Z 684.904,A -85,B 0,C 180,E1 -19016.559,E2 -19016.559} C_VEL
LIN {X 0,Y 264.472,Z 672.541,A -85,B 0,C 180,E1 -19017.389,E2 -19017.389} C_VEL
LIN {X 0,Y 265.397,Z 659.703,A -85,B 0,C 180,E1 -19017.928,E2 -19017.928} C_VEL
LIN {X 0,Y 267.425,Z 595.25,A -85,B 0,C 180,E1 -19019.651,E2 -19019.651} C_VEL
LIN {X 0,Y 260.981,Z 579.13,A -85,B 0,C 180,E1 -19020.972,E2 -19020.972} C_VEL
LIN {X 0,Y 253.284,Z 563.062,A -85,B 0,C 180,E1 -19022.559,E2 -19022.559} C_VEL
LIN {X 0,Y 249.649,Z 555.829,A -85,B 0,C 180,E1 -19023.404,E2 -19023.404} C_VEL
LIN {X 0,Y 249.109,Z 553.695,A -85,B 0,C 180,E1 -19024.348,E2 -19024.348} C_VEL
LIN {X 0,Y 249.067,Z 553.451,A -85,B 0,C 180,E1 -19026.337,E2 -19026.337} C_VEL
LIN {X 0,Y 249.022,Z 553.452,A -85,B 0,C 180,E1 -19030.473,E2 -19030.473} C_VEL
LIN {X 0,Y 249.001,Z 553.446,A -85,B 0,C 180,E1 -19034.877,E2 -19034.877} C_VEL
LIN {X 0,Y 249.023,Z 553.464,A -85,B 0,C 180,E1 -19037.364,E2 -19037.364} C_VEL
LIN {X 0,Y 249.046,Z 553.431,A -85,B 0,C 180,E1 -19041.623,E2 -19041.623} C_VEL
LIN {X 0,Y 249.057,Z 553.463,A -85,B 0,C 180,E1 -19045.641,E2 -19045.641} C_VEL
LIN {X 0,Y 249.047,Z 553.463,A -85,B 0,C 180,E1 -19049.472,E2 -19049.472} C_VEL
LIN {X 0,Y 249.068,Z 553.449,A -85,B 0,C 180,E1 -19053.161,E2 -19053.161} C_VEL
LIN {X 0,Y 249.073,Z 553.451,A -85,B 0,C 180,E1 -19056.732,E2 -19056.732} C_VEL
LIN {X 0,Y 249.105,Z 553.454,A -85,B 0,C 180,E1 -19060.211,E2 -19060.211} C_VEL
LIN {X 0,Y 249.191,Z 553.428,A -85,B 0,C 180,E1 -19064.457,E2 -19064.457} C_VEL
LIN {X 0,Y 248.516,Z 553.524,A -85,B 0,C 180,E1 -19065.806,E2 -19065.806} C_VEL
LIN {X 0,Y 245.707,Z 553.874,A -85,B 0,C 180,E1 -19068.007,E2 -19068.007} C_VEL
LIN {X 0,Y 243.384,Z 554.153,A -85,B 0,C 180,E1 -19069.8,E2 -19069.8} C_VEL
LIN {X 0,Y 242.459,Z 554.268,A -85,B 0,C 180,E1 -19071.189,E2 -19071.189} C_VEL
LIN {X 0,Y 242.42,Z 554.277,A -85,B 0,C 180,E1 -19071.658,E2 -19071.658} C_VEL
LIN {X 0,Y 242.255,Z 554.303,A -85,B 0,C 180,E1 -19075.007,E2 -19075.007} C_VEL
LIN {X 0,Y 242.63,Z 554.252,A -85,B 0,C 180,E1 -19078.34,E2 -19078.34} C_VEL
LIN {X 0,Y 242.631,Z 554.256,A -85,B 0,C 180,E1 -19081.66,E2 -19081.66} C_VEL
LIN {X 0,Y 242.428,Z 554.286,A -85,B 0,C 180,E1 -19086.659,E2 -19086.659} C_VEL
LIN {X 0,Y 242.339,Z 554.28,A -85,B 0,C 180,E1 -19090.021,E2 -19090.021} C_VEL
LIN {X 0,Y 242.161,Z 554.31,A -85,B 0,C 180,E1 -19095.141,E2 -19095.141} C_VEL
LIN {X 0,Y 242.068,Z 554.331,A -85,B 0,C 180,E1 -19098.625,E2 -19098.625} C_VEL
LIN {X 0,Y 242.007,Z 554.328,A -85,B 0,C 180,E1 -19102.181,E2 -19102.181} C_VEL
LIN {X 0,Y 242.06,Z 554.324,A -85,B 0,C 180,E1 -19105.839,E2 -19105.839} C_VEL
LIN {X 0,Y 242.001,Z 554.339,A -85,B 0,C 180,E1 -19109.584,E2 -19109.584} C_VEL
LIN {X 0,Y 241.975,Z 554.344,A -85,B 0,C 180,E1 -19113.494,E2 -19113.494} C_VEL
LIN {X 0,Y 241.985,Z 554.317,A -85,B 0,C 180,E1 -19117.583,E2 -19117.583} C_VEL
LIN {X 0,Y 241.951,Z 554.328,A -85,B 0,C 180,E1 -19121.92,E2 -19121.92} C_VEL
LIN {X 0,Y 241.998,Z 554.328,A -85,B 0,C 180,E1 -19126.556,E2 -19126.556} C_VEL
LIN {X 0,Y 242.066,Z 554.398,A -85,B 0,C 180,E1 -19130.063,E2 -19130.063} C_VEL
LIN {X 0,Y 243.966,Z 562.14,A -85,B 0,C 180,E1 -19133.766,E2 -19133.766} C_VEL
LIN {X 0,Y 245.178,Z 567.218,A -85,B 0,C 180,E1 -19135.926,E2 -19135.926} C_VEL
LIN {X 0,Y 248.049,Z 573.648,A -85,B 0,C 180,E1 -19136.658,E2 -19136.658} C_VEL
LIN {X 0,Y 254.453,Z 587.836,A -85,B 0,C 180,E1 -19138.058,E2 -19138.058} C_VEL
LIN {X 0,Y 257.27,Z 595.421,A -85,B 0,C 180,E1 -19138.688,E2 -19138.688} C_VEL
LIN {X 0,Y 260.635,Z 618.502,A -85,B 0,C 180,E1 -19139.856,E2 -19139.856} C_VEL
LIN {X 0,Y 258.548,Z 675.97,A -85,B 0,C 180,E1 -19141.431,E2 -19141.431} C_VEL
LIN {X 0,Y 257.3,Z 689.856,A -85,B 0,C 180,E1 -19142.113,E2 -19142.113} C_VEL
LIN {X 0,Y 255.684,Z 702.294,A -85,B 0,C 180,E1 -19143.031,E2 -19143.031} C_VEL
LIN {X 0,Y 253.908,Z 713.401,A -85,B 0,C 180,E1 -19144.156,E2 -19144.156} C_VEL
LIN {X 0,Y 251.665,Z 724.966,A -85,B 0,C 180,E1 -19145.677,E2 -19145.677} C_VEL
LIN {X 0,Y 249.409,Z 735.383,A -85,B 0,C 180,E1 -19147.424,E2 -19147.424} C_VEL
LIN {X 0,Y 247.45,Z 743.906,A -85,B 0,C 180,E1 -19149.207,E2 -19149.207} C_VEL
LIN {X 0,Y 245.289,Z 753.148,A -85,B 0,C 180,E1 -19151.63,E2 -19151.63} C_VEL
LIN {X 0,Y 243.378,Z 760.577,A -85,B 0,C 180,E1 -19154.079,E2 -19154.079} C_VEL
LIN {X 0,Y 241.836,Z 766.542,A -85,B 0,C 180,E1 -19156.558,E2 -19156.558} C_VEL
LIN {X 0,Y 240.859,Z 771.264,A -85,B 0,C 180,E1 -19159.068,E2 -19159.068} C_VEL
LIN {X 0,Y 240.214,Z 774.877,A -85,B 0,C 180,E1 -19161.59,E2 -19161.59} C_VEL
LIN {X 0,Y 239.951,Z 776.74,A -85,B 0,C 180,E1 -19163.273,E2 -19163.273} C_VEL
LIN {X 0,Y 239.773,Z 778.339,A -85,B 0,C 180,E1 -19165.258,E2 -19165.258} C_VEL
LIN {X 0,Y 239.812,Z 779.744,A -85,B 0,C 180,E1 -19168.322,E2 -19168.322} C_VEL
LIN {X 0,Y 239.888,Z 779.875,A -85,B 0,C 180,E1 -19171.47,E2 -19171.47} C_VEL
LIN {X 0,Y 239.893,Z 781.754,A -85,B 0,C 180,E1 -19173.36,E2 -19173.36} C_VEL
LIN {X 0,Y 239.992,Z 782.984,A -85,B 0,C 180,E1 -19175.335,E2 -19175.335} C_VEL
LIN {X 0,Y 240.52,Z 783.518,A -85,B 0,C 180,E1 -19178.402,E2 -19178.402} C_VEL
LIN {X 0,Y 241.164,Z 783.128,A -85,B 0,C 180,E1 -19180.071,E2 -19180.071} C_VEL
LIN {X 0,Y 241.986,Z 782.154,A -85,B 0,C 180,E1 -19181.731,E2 -19181.731} C_VEL
LIN {X 0,Y 242.966,Z 780.691,A -85,B 0,C 180,E1 -19183.381,E2 -19183.381} C_VEL
LIN {X 0,Y 244.803,Z 777.564,A -85,B 0,C 180,E1 -19185.828,E2 -19185.828} C_VEL
LIN {X 0,Y 247.289,Z 773.197,A -85,B 0,C 180,E1 -19188.219,E2 -19188.219} C_VEL
LIN {X 0,Y 250.18,Z 767.252,A -85,B 0,C 180,E1 -19190.559,E2 -19190.559} C_VEL
LIN {X 0,Y 252.849,Z 761.15,A -85,B 0,C 180,E1 -19192.47,E2 -19192.47} C_VEL
LIN {X 0,Y 255.779,Z 753.729,A -85,B 0,C 180,E1 -19194.341,E2 -19194.341} C_VEL
LIN {X 0,Y 259.48,Z 743.381,A -85,B 0,C 180,E1 -19196.33,E2 -19196.33} C_VEL
LIN {X 0,Y 262.002,Z 735.351,A -85,B 0,C 180,E1 -19197.564,E2 -19197.564} C_VEL
LIN {X 0,Y 264.707,Z 725.401,A -85,B 0,C 180,E1 -19198.798,E2 -19198.798} C_VEL
LIN {X 0,Y 267.263,Z 714.077,A -85,B 0,C 180,E1 -19199.868,E2 -19199.868} C_VEL
LIN {X 0,Y 269.256,Z 702.524,A -85,B 0,C 180,E1 -19200.706,E2 -19200.706} C_VEL
LIN {X 0,Y 274.43,Z 668.532,A -85,B 0,C 180,E1 -19202.481,E2 -19202.481} C_VEL
LIN {X 0,Y 281.297,Z 626.742,A -85,B 0,C 180,E1 -19204.525,E2 -19204.525} C_VEL
LIN {X 0,Y 281.466,Z 622.311,A -85,B 0,C 180,E1 -19205.026,E2 -19205.026} C_VEL
LIN {X 0,Y 280.498,Z 619.783,A -85,B 0,C 180,E1 -19205.894,E2 -19205.894} C_VEL
LIN {X 0,Y 278.931,Z 617.731,A -85,B 0,C 180,E1 -19207.209,E2 -19207.209} C_VEL
LIN {X 0,Y 277.431,Z 615.891,A -85,B 0,C 180,E1 -19209.296,E2 -19209.296} C_VEL
LIN {X 0,Y 276.334,Z 614.937,A -85,B 0,C 180,E1 -19211.397,E2 -19211.397} C_VEL
LIN {X 0,Y 275.295,Z 614.922,A -85,B 0,C 180,E1 -19214.372,E2 -19214.372} C_VEL
LIN {X 0,Y 274.885,Z 615.785,A -85,B 0,C 180,E1 -19216.345,E2 -19216.345} C_VEL
LIN {X 0,Y 274.686,Z 618.134,A -85,B 0,C 180,E1 -19219.123,E2 -19219.123} C_VEL
LIN {X 0,Y 275.923,Z 622.423,A -85,B 0,C 180,E1 -19221.527,E2 -19221.527} C_VEL
LIN {X 0,Y 276.984,Z 625.736,A -85,B 0,C 180,E1 -19222.903,E2 -19222.903} C_VEL
LIN {X 0,Y 277.643,Z 628.423,A -85,B 0,C 180,E1 -19223.75,E2 -19223.75} C_VEL
LIN {X 0,Y 278.249,Z 641.035,A -85,B 0,C 180,E1 -19225.823,E2 -19225.823} C_VEL
LIN {X 0,Y 278.845,Z 653.763,A -85,B 0,C 180,E1 -19227.563,E2 -19227.563} C_VEL
LIN {X 0,Y 278.893,Z 661.315,A -85,B 0,C 180,E1 -19228.397,E2 -19228.397} C_VEL
LIN {X 0,Y 272.611,Z 702.728,A -85,B 0,C 180,E1 -19230.406,E2 -19230.406} C_VEL
LIN {X 0,Y 270.127,Z 714.863,A -85,B 0,C 180,E1 -19231.228,E2 -19231.228} C_VEL
LIN {X 0,Y 267.49,Z 725.131,A -85,B 0,C 180,E1 -19232.202,E2 -19232.202} C_VEL
LIN {X 0,Y 264.558,Z 734.74,A -85,B 0,C 180,E1 -19233.366,E2 -19233.366} C_VEL
LIN {X 0,Y 261.033,Z 744.672,A -85,B 0,C 180,E1 -19234.909,E2 -19234.909} C_VEL
LIN {X 0,Y 258.108,Z 751.893,A -85,B 0,C 180,E1 -19236.32,E2 -19236.32} C_VEL
LIN {X 0,Y 255.416,Z 757.941,A -85,B 0,C 180,E1 -19237.769,E2 -19237.769} C_VEL
LIN {X 0,Y 252.36,Z 764.151,A -85,B 0,C 180,E1 -19239.628,E2 -19239.628} C_VEL
LIN {X 0,Y 249.207,Z 770.133,A -85,B 0,C 180,E1 -19241.928,E2 -19241.928} C_VEL
LIN {X 0,Y 246.423,Z 774.571,A -85,B 0,C 180,E1 -19244.28,E2 -19244.28} C_VEL
LIN {X 0,Y 244.129,Z 777.648,A -85,B 0,C 180,E1 -19246.685,E2 -19246.685} C_VEL
LIN {X 0,Y 242.929,Z 779.1,A -85,B 0,C 180,E1 -19248.316,E2 -19248.316} C_VEL
LIN {X 0,Y 241.937,Z 780.028,A -85,B 0,C 180,E1 -19249.963,E2 -19249.963} C_VEL
LIN {X 0,Y 241.211,Z 780.363,A -85,B 0,C 180,E1 -19251.623,E2 -19251.623} C_VEL
LIN {X 0,Y 240.624,Z 780.211,A -85,B 0,C 180,E1 -19253.291,E2 -19253.291} C_VEL
LIN {X 0,Y 240.18,Z 779.588,A -85,B 0,C 180,E1 -19254.964,E2 -19254.964} C_VEL
LIN {X 0,Y 239.956,Z 778.468,A -85,B 0,C 180,E1 -19256.642,E2 -19256.642} C_VEL
LIN {X 0,Y 239.87,Z 775.656,A -85,B 0,C 180,E1 -19259.161,E2 -19259.161} C_VEL
LIN {X 0,Y 239.934,Z 771.56,A -85,B 0,C 180,E1 -19261.679,E2 -19261.679} C_VEL
LIN {X 0,Y 240.116,Z 768,A -85,B 0,C 180,E1 -19263.356,E2 -19263.356} C_VEL
LIN {X 0,Y 240.294,Z 762.714,A -85,B 0,C 180,E1 -19265.366,E2 -19265.366} C_VEL
LIN {X 0,Y 240.678,Z 755.492,A -85,B 0,C 180,E1 -19267.551,E2 -19267.551} C_VEL
LIN {X 0,Y 241.045,Z 748.523,A -85,B 0,C 180,E1 -19269.228,E2 -19269.228} C_VEL
LIN {X 0,Y 241.548,Z 740.057,A -85,B 0,C 180,E1 -19270.902,E2 -19270.902} C_VEL
LIN {X 0,Y 242.122,Z 731.023,A -85,B 0,C 180,E1 -19272.361,E2 -19272.361} C_VEL
LIN {X 0,Y 242.846,Z 719.452,A -85,B 0,C 180,E1 -19273.813,E2 -19273.813} C_VEL
LIN {X 0,Y 243.358,Z 708.405,A -85,B 0,C 180,E1 -19274.851,E2 -19274.851} C_VEL
LIN {X 0,Y 243.794,Z 694.903,A -85,B 0,C 180,E1 -19275.733,E2 -19275.733} C_VEL
LIN {X 0,Y 245.236,Z 644.331,A -85,B 0,C 180,E1 -19278.159,E2 -19278.159} C_VEL
LIN {X 0,Y 243.522,Z 621.09,A -85,B 0,C 180,E1 -19279.296,E2 -19279.296} C_VEL
LIN {X 0,Y 243.495,Z 617.23,A -85,B 0,C 180,E1 -19279.539,E2 -19279.539} C_VEL
LIN {X 0,Y 245.163,Z 597.85,A -85,B 0,C 180,E1 -19284.111,E2 -19284.111} C_VEL
LIN {X 0,Y 246.928,Z 579.712,A -85,B 0,C 180,E1 -19288.386,E2 -19288.386} C_VEL
LIN {X 0,Y 246.412,Z 575.299,A -85,B 0,C 180,E1 -19289.472,E2 -19289.472} C_VEL
LIN {X 0,Y 242.435,Z 555.922,A -85,B 0,C 180,E1 -19294.423,E2 -19294.423} C_VEL
LIN {X 0,Y 242.134,Z 554.445,A -85,B 0,C 180,E1 -19294.914,E2 -19294.914} C_VEL
LIN {X 0,Y 241.977,Z 554.308,A -85,B 0,C 180,E1 -19299.715,E2 -19299.715} C_VEL
LIN {X 0,Y 241.927,Z 554.303,A -85,B 0,C 180,E1 -19304.203,E2 -19304.203} C_VEL
LIN {X 0,Y 241.938,Z 554.327,A -85,B 0,C 180,E1 -19308.076,E2 -19308.076} C_VEL
LIN {X 0,Y 241.993,Z 554.319,A -85,B 0,C 180,E1 -19312.417,E2 -19312.417} C_VEL
LIN {X 0,Y 242.05,Z 554.502,A -85,B 0,C 180,E1 -19314.915,E2 -19314.915} C_VEL
LIN {X 0,Y 242.493,Z 556.177,A -85,B 0,C 180,E1 -19315.629,E2 -19315.629} C_VEL
LIN {X 0,Y 250.254,Z 571.289,A -85,B 0,C 180,E1 -19317.406,E2 -19317.406} C_VEL
LIN {X 0,Y 257.285,Z 586.85,A -85,B 0,C 180,E1 -19318.91,E2 -19318.91} C_VEL
LIN {X 0,Y 261.208,Z 596.939,A -85,B 0,C 180,E1 -19319.748,E2 -19319.748} C_VEL
LIN {X 0,Y 258.9,Z 662.781,A -85,B 0,C 180,E1 -19321.554,E2 -19321.554} C_VEL
LIN {X 0,Y 257.788,Z 676.351,A -85,B 0,C 180,E1 -19322.227,E2 -19322.227} C_VEL
LIN {X 0,Y 256.287,Z 689.349,A -85,B 0,C 180,E1 -19323.207,E2 -19323.207} C_VEL
LIN {X 0,Y 254.494,Z 701.144,A -85,B 0,C 180,E1 -19324.436,E2 -19324.436} C_VEL
LIN {X 0,Y 252.438,Z 712.484,A -85,B 0,C 180,E1 -19325.972,E2 -19325.972} C_VEL
LIN {X 0,Y 250.184,Z 723.103,A -85,B 0,C 180,E1 -19327.799,E2 -19327.799} C_VEL
LIN {X 0,Y 248.332,Z 731.863,A -85,B 0,C 180,E1 -19329.714,E2 -19329.714} C_VEL
LIN {X 0,Y 246.012,Z 740.772,A -85,B 0,C 180,E1 -19332.114,E2 -19332.114} C_VEL
LIN {X 0,Y 244.156,Z 747.937,A -85,B 0,C 180,E1 -19334.557,E2 -19334.557} C_VEL
LIN {X 0,Y 242.864,Z 752.77,A -85,B 0,C 180,E1 -19336.613,E2 -19336.613} C_VEL
LIN {X 0,Y 241.618,Z 757.464,A -85,B 0,C 180,E1 -19339.1,E2 -19339.1} C_VEL
LIN {X 0,Y 240.808,Z 761.049,A -85,B 0,C 180,E1 -19341.608,E2 -19341.608} C_VEL
LIN {X 0,Y 240.32,Z 763.43,A -85,B 0,C 180,E1 -19343.888,E2 -19343.888} C_VEL
LIN {X 0,Y 240.036,Z 765.283,A -85,B 0,C 180,E1 -19346.642,E2 -19346.642} C_VEL
LIN {X 0,Y 239.924,Z 766.122,A -85,B 0,C 180,E1 -19349.999,E2 -19349.999} C_VEL
LIN {X 0,Y 239.919,Z 765.93,A -85,B 0,C 180,E1 -19351.677,E2 -19351.677} C_VEL
LIN {X 0,Y 240.033,Z 765.345,A -85,B 0,C 180,E1 -19353.356,E2 -19353.356} C_VEL
LIN {X 0,Y 240.449,Z 763.025,A -85,B 0,C 180,E1 -19356.713,E2 -19356.713} C_VEL
LIN {X 0,Y 241.037,Z 760.157,A -85,B 0,C 180,E1 -19359.227,E2 -19359.227} C_VEL
LIN {X 0,Y 241.963,Z 756.265,A -85,B 0,C 180,E1 -19361.73,E2 -19361.73} C_VEL
LIN {X 0,Y 243.288,Z 751.247,A -85,B 0,C 180,E1 -19364.212,E2 -19364.212} C_VEL
LIN {X 0,Y 244.885,Z 744.927,A -85,B 0,C 180,E1 -19366.676,E2 -19366.676} C_VEL
LIN {X 0,Y 247.048,Z 737.009,A -85,B 0,C 180,E1 -19369.094,E2 -19369.094} C_VEL
LIN {X 0,Y 249.189,Z 728.144,A -85,B 0,C 180,E1 -19371.268,E2 -19371.268} C_VEL
LIN {X 0,Y 251.318,Z 717.997,A -85,B 0,C 180,E1 -19373.264,E2 -19373.264} C_VEL
LIN {X 0,Y 253.59,Z 706.587,A -85,B 0,C 180,E1 -19375,E2 -19375} C_VEL
LIN {X 0,Y 255.586,Z 695.366,A -85,B 0,C 180,E1 -19376.319,E2 -19376.319} C_VEL
LIN {X 0,Y 257.103,Z 683.964,A -85,B 0,C 180,E1 -19377.358,E2 -19377.358} C_VEL
LIN {X 0,Y 258.36,Z 670.914,A -85,B 0,C 180,E1 -19378.204,E2 -19378.204} C_VEL
LIN {X 0,Y 259.235,Z 658.384,A -85,B 0,C 180,E1 -19378.707,E2 -19378.707} C_VEL
LIN {X 0,Y 261.26,Z 597.047,A -85,B 0,C 180,E1 -19380.373,E2 -19380.373} C_VEL
LIN {X 0,Y 254.882,Z 581.211,A -85,B 0,C 180,E1 -19381.737,E2 -19381.737} C_VEL
LIN {X 0,Y 247.507,Z 565.943,A -85,B 0,C 180,E1 -19383.325,E2 -19383.325} C_VEL
LIN {X 0,Y 242.475,Z 556.117,A -85,B 0,C 180,E1 -19384.519,E2 -19384.519} C_VEL
LIN {X 0,Y 242.038,Z 554.426,A -85,B 0,C 180,E1 -19385.319,E2 -19385.319} C_VEL
LIN {X 0,Y 241.969,Z 554.329,A -85,B 0,C 180,E1 -19389.714,E2 -19389.714} C_VEL
LIN {X 0,Y 241.928,Z 554.329,A -85,B 0,C 180,E1 -19394.2,E2 -19394.2} C_VEL
LIN {X 0,Y 241.95,Z 554.347,A -85,B 0,C 180,E1 -19398.08,E2 -19398.08} C_VEL
LIN {X 0,Y 242.007,Z 554.311,A -85,B 0,C 180,E1 -19402.421,E2 -19402.421} C_VEL
LIN {X 0,Y 241.986,Z 554.339,A -85,B 0,C 180,E1 -19406.508,E2 -19406.508} C_VEL
LIN {X 0,Y 242.031,Z 554.336,A -85,B 0,C 180,E1 -19410.586,E2 -19410.586} C_VEL
LIN {X 0,Y 242.062,Z 554.332,A -85,B 0,C 180,E1 -19414.182,E2 -19414.182} C_VEL
LIN {X 0,Y 242.047,Z 554.32,A -85,B 0,C 180,E1 -19418.296,E2 -19418.296} C_VEL
LIN {X 0,Y 242.157,Z 554.305,A -85,B 0,C 180,E1 -19423.278,E2 -19423.278} C_VEL
LIN {X 0,Y 242.18,Z 554.312,A -85,B 0,C 180,E1 -19428.279,E2 -19428.279} C_VEL
LIN {X 0,Y 242.42,Z 554.277,A -85,B 0,C 180,E1 -19431.658,E2 -19431.658} C_VEL
LIN {X 0,Y 241.859,Z 554.359,A -85,B 0,C 180,E1 -19433.043,E2 -19433.043} C_VEL
LIN {X 0,Y 239.077,Z 554.701,A -85,B 0,C 180,E1 -19435.303,E2 -19435.303} C_VEL
LIN {X 0,Y 236.672,Z 554.993,A -85,B 0,C 180,E1 -19437.145,E2 -19437.145} C_VEL
LIN {X 0,Y 235.661,Z 555.122,A -85,B 0,C 180,E1 -19438.574,E2 -19438.574} C_VEL
LIN {X 0,Y 235.593,Z 555.129,A -85,B 0,C 180,E1 -19439.058,E2 -19439.058} C_VEL
LIN {X 0,Y 235.59,Z 555.132,A -85,B 0,C 180,E1 -19441.709,E2 -19441.709} C_VEL
LIN {X 0,Y 235.4,Z 555.162,A -85,B 0,C 180,E1 -19446.859,E2 -19446.859} C_VEL
LIN {X 0,Y 235.247,Z 555.164,A -85,B 0,C 180,E1 -19450.326,E2 -19450.326} C_VEL
LIN {X 0,Y 235.108,Z 555.184,A -85,B 0,C 180,E1 -19455.607,E2 -19455.607} C_VEL
LIN {X 0,Y 235.003,Z 555.213,A -85,B 0,C 180,E1 -19459.206,E2 -19459.206} C_VEL
LIN {X 0,Y 234.955,Z 555.212,A -85,B 0,C 180,E1 -19462.883,E2 -19462.883} C_VEL
LIN {X 0,Y 234.961,Z 555.205,A -85,B 0,C 180,E1 -19466.658,E2 -19466.658} C_VEL
LIN {X 0,Y 234.916,Z 555.216,A -85,B 0,C 180,E1 -19470.57,E2 -19470.57} C_VEL
LIN {X 0,Y 234.921,Z 555.208,A -85,B 0,C 180,E1 -19474.64,E2 -19474.64} C_VEL
LIN {X 0,Y 234.937,Z 555.215,A -85,B 0,C 180,E1 -19478.946,E2 -19478.946} C_VEL
LIN {X 0,Y 234.922,Z 555.206,A -85,B 0,C 180,E1 -19483.478,E2 -19483.478} C_VEL
LIN {X 0,Y 234.97,Z 555.203,A -85,B 0,C 180,E1 -19486.536,E2 -19486.536} C_VEL
LIN {X 0,Y 234.97,Z 555.249,A -85,B 0,C 180,E1 -19489.065,E2 -19489.065} C_VEL
LIN {X 0,Y 236.1,Z 559.501,A -85,B 0,C 180,E1 -19491.312,E2 -19491.312} C_VEL
LIN {X 0,Y 237.92,Z 567.072,A -85,B 0,C 180,E1 -19494.753,E2 -19494.753} C_VEL
LIN {X 0,Y 245.327,Z 582.799,A -85,B 0,C 180,E1 -19496.557,E2 -19496.557} C_VEL
LIN {X 0,Y 251.265,Z 597.038,A -85,B 0,C 180,E1 -19497.911,E2 -19497.911} C_VEL
LIN {X 0,Y 254.495,Z 619.574,A -85,B 0,C 180,E1 -19499.09,E2 -19499.09} C_VEL
LIN {X 0,Y 252.341,Z 675.779,A -85,B 0,C 180,E1 -19500.661,E2 -19500.661} C_VEL
LIN {X 0,Y 251.067,Z 689.661,A -85,B 0,C 180,E1 -19501.357,E2 -19501.357} C_VEL
LIN {X 0,Y 249.379,Z 702.095,A -85,B 0,C 180,E1 -19502.291,E2 -19502.291} C_VEL
LIN {X 0,Y 247.544,Z 713.201,A -85,B 0,C 180,E1 -19503.44,E2 -19503.44} C_VEL
LIN {X 0,Y 245.212,Z 724.765,A -85,B 0,C 180,E1 -19504.994,E2 -19504.994} C_VEL
LIN {X 0,Y 242.839,Z 735.181,A -85,B 0,C 180,E1 -19506.778,E2 -19506.778} C_VEL
LIN {X 0,Y 240.801,Z 743.704,A -85,B 0,C 180,E1 -19508.605,E2 -19508.605} C_VEL
LIN {X 0,Y 238.944,Z 751.457,A -85,B 0,C 180,E1 -19510.644,E2 -19510.644} C_VEL
LIN {X 0,Y 236.853,Z 759.253,A -85,B 0,C 180,E1 -19513.185,E2 -19513.185} C_VEL
LIN {X 0,Y 234.896,Z 766.338,A -85,B 0,C 180,E1 -19516.153,E2 -19516.153} C_VEL
LIN {X 0,Y 233.875,Z 771.06,A -85,B 0,C 180,E1 -19518.738,E2 -19518.738} C_VEL
LIN {X 0,Y 233.181,Z 774.673,A -85,B 0,C 180,E1 -19521.334,E2 -19521.334} C_VEL
LIN {X 0,Y 232.889,Z 776.536,A -85,B 0,C 180,E1 -19523.068,E2 -19523.068} C_VEL
LIN {X 0,Y 232.684,Z 778.303,A -85,B 0,C 180,E1 -19525.37,E2 -19525.37} C_VEL
LIN {X 0,Y 232.726,Z 779.539,A -85,B 0,C 180,E1 -19528.271,E2 -19528.271} C_VEL
LIN {X 0,Y 232.774,Z 779.753,A -85,B 0,C 180,E1 -19530.001,E2 -19530.001} C_VEL
LIN {X 0,Y 232.824,Z 779.588,A -85,B 0,C 180,E1 -19531.948,E2 -19531.948} C_VEL
LIN {X 0,Y 232.842,Z 781.099,A -85,B 0,C 180,E1 -19533.462,E2 -19533.462} C_VEL
LIN {X 0,Y 232.914,Z 782.45,A -85,B 0,C 180,E1 -19535.283,E2 -19535.283} C_VEL
LIN {X 0,Y 233.087,Z 783.217,A -85,B 0,C 180,E1 -19536.929,E2 -19536.929} C_VEL
LIN {X 0,Y 233.496,Z 783.501,A -85,B 0,C 180,E1 -19538.657,E2 -19538.657} C_VEL
LIN {X 0,Y 234.159,Z 783.217,A -85,B 0,C 180,E1 -19540.376,E2 -19540.376} C_VEL
LIN {X 0,Y 235.046,Z 782.471,A -85,B 0,C 180,E1 -19542.083,E2 -19542.083} C_VEL
LIN {X 0,Y 236.097,Z 781.272,A -85,B 0,C 180,E1 -19543.778,E2 -19543.778} C_VEL
LIN {X 0,Y 238.042,Z 778.461,A -85,B 0,C 180,E1 -19546.29,E2 -19546.29} C_VEL
LIN {X 0,Y 240.665,Z 774.397,A -85,B 0,C 180,E1 -19548.738,E2 -19548.738} C_VEL
LIN {X 0,Y 243.741,Z 769.085,A -85,B 0,C 180,E1 -19551.128,E2 -19551.128} C_VEL
LIN {X 0,Y 247.19,Z 762.069,A -85,B 0,C 180,E1 -19553.457,E2 -19553.457} C_VEL
LIN {X 0,Y 250.366,Z 754.908,A -85,B 0,C 180,E1 -19555.347,E2 -19555.347} C_VEL
LIN {X 0,Y 253.604,Z 747.05,A -85,B 0,C 180,E1 -19556.989,E2 -19556.989} C_VEL
LIN {X 0,Y 257.267,Z 736.656,A -85,B 0,C 180,E1 -19558.694,E2 -19558.694} C_VEL
LIN {X 0,Y 260.281,Z 726.789,A -85,B 0,C 180,E1 -19559.97,E2 -19559.97} C_VEL
LIN {X 0,Y 263.327,Z 714.757,A -85,B 0,C 180,E1 -19561.139,E2 -19561.139} C_VEL
LIN {X 0,Y 265.586,Z 702.957,A -85,B 0,C 180,E1 -19562.012,E2 -19562.012} C_VEL
LIN {X 0,Y 271.065,Z 669.771,A -85,B 0,C 180,E1 -19563.768,E2 -19563.768} C_VEL
LIN {X 0,Y 278.339,Z 628.738,A -85,B 0,C 180,E1 -19565.792,E2 -19565.792} C_VEL
LIN {X 0,Y 278.384,Z 626.891,A -85,B 0,C 180,E1 -19566.028,E2 -19566.028} C_VEL
LIN {X 0,Y 277.388,Z 625.119,A -85,B 0,C 180,E1 -19566.918,E2 -19566.918} C_VEL
LIN {X 0,Y 274.955,Z 622.584,A -85,B 0,C 180,E1 -19569.262,E2 -19569.262} C_VEL
LIN {X 0,Y 273.185,Z 621.318,A -85,B 0,C 180,E1 -19571.75,E2 -19571.75} C_VEL
LIN {X 0,Y 272.29,Z 621.285,A -85,B 0,C 180,E1 -19574.179,E2 -19574.179} C_VEL
LIN {X 0,Y 272.149,Z 622.757,A -85,B 0,C 180,E1 -19576.773,E2 -19576.773} C_VEL
LIN {X 0,Y 272.727,Z 624.963,A -85,B 0,C 180,E1 -19578.916,E2 -19578.916} C_VEL
LIN {X 0,Y 273.933,Z 629.363,A -85,B 0,C 180,E1 -19581.339,E2 -19581.339} C_VEL
LIN {X 0,Y 274.89,Z 633.234,A -85,B 0,C 180,E1 -19582.819,E2 -19582.819} C_VEL
LIN {X 0,Y 275.112,Z 645.523,A -85,B 0,C 180,E1 -19584.878,E2 -19584.878} C_VEL
LIN {X 0,Y 275.3,Z 657.428,A -85,B 0,C 180,E1 -19586.533,E2 -19586.533} C_VEL
LIN {X 0,Y 275.257,Z 663.063,A -85,B 0,C 180,E1 -19587.17,E2 -19587.17} C_VEL
LIN {X 0,Y 268.54,Z 704.014,A -85,B 0,C 180,E1 -19589.205,E2 -19589.205} C_VEL
LIN {X 0,Y 265.8,Z 716.199,A -85,B 0,C 180,E1 -19590.061,E2 -19590.061} C_VEL
LIN {X 0,Y 263.018,Z 726.068,A -85,B 0,C 180,E1 -19591.033,E2 -19591.033} C_VEL
LIN {X 0,Y 259.461,Z 736.699,A -85,B 0,C 180,E1 -19592.363,E2 -19592.363} C_VEL
LIN {X 0,Y 255.763,Z 746.171,A -85,B 0,C 180,E1 -19593.918,E2 -19593.918} C_VEL
LIN {X 0,Y 252.638,Z 753.111,A -85,B 0,C 180,E1 -19595.337,E2 -19595.337} C_VEL
LIN {X 0,Y 249.101,Z 760.255,A -85,B 0,C 180,E1 -19597.174,E2 -19597.174} C_VEL
LIN {X 0,Y 245.937,Z 766.121,A -85,B 0,C 180,E1 -19599.071,E2 -19599.071} C_VEL
LIN {X 0,Y 242.588,Z 771.523,A -85,B 0,C 180,E1 -19601.417,E2 -19601.417} C_VEL
LIN {X 0,Y 239.68,Z 775.55,A -85,B 0,C 180,E1 -19603.826,E2 -19603.826} C_VEL
LIN {X 0,Y 238.791,Z 776.692,A -85,B 0,C 180,E1 -19604.64,E2 -19604.64} C_VEL
LIN {X 0,Y 237.273,Z 778.368,A -85,B 0,C 180,E1 -19606.293,E2 -19606.293} C_VEL
LIN {X 0,Y 235.994,Z 779.546,A -85,B 0,C 180,E1 -19607.968,E2 -19607.968} C_VEL
LIN {X 0,Y 234.971,Z 780.256,A -85,B 0,C 180,E1 -19609.662,E2 -19609.662} C_VEL
LIN {X 0,Y 234.187,Z 780.496,A -85,B 0,C 180,E1 -19611.37,E2 -19611.37} C_VEL
LIN {X 0,Y 233.532,Z 780.104,A -85,B 0,C 180,E1 -19613.282,E2 -19613.282} C_VEL
LIN {X 0,Y 232.911,Z 777.947,A -85,B 0,C 180,E1 -19616.54,E2 -19616.54} C_VEL
LIN {X 0,Y 232.807,Z 774.917,A -85,B 0,C 180,E1 -19619.135,E2 -19619.135} C_VEL
LIN {X 0,Y 232.892,Z 770.559,A -85,B 0,C 180,E1 -19621.729,E2 -19621.729} C_VEL
LIN {X 0,Y 233.189,Z 764.519,A -85,B 0,C 180,E1 -19624.321,E2 -19624.321} C_VEL
LIN {X 0,Y 233.427,Z 759.095,A -85,B 0,C 180,E1 -19626.168,E2 -19626.168} C_VEL
LIN {X 0,Y 233.757,Z 751.741,A -85,B 0,C 180,E1 -19628.211,E2 -19628.211} C_VEL
LIN {X 0,Y 234.335,Z 741.929,A -85,B 0,C 180,E1 -19630.367,E2 -19630.367} C_VEL
LIN {X 0,Y 234.928,Z 733.249,A -85,B 0,C 180,E1 -19631.869,E2 -19631.869} C_VEL
LIN {X 0,Y 235.545,Z 722.456,A -85,B 0,C 180,E1 -19633.37,E2 -19633.37} C_VEL
LIN {X 0,Y 236.141,Z 711.102,A -85,B 0,C 180,E1 -19634.544,E2 -19634.544} C_VEL
LIN {X 0,Y 236.491,Z 699.774,A -85,B 0,C 180,E1 -19635.403,E2 -19635.403} C_VEL
LIN {X 0,Y 238.042,Z 651.129,A -85,B 0,C 180,E1 -19637.884,E2 -19637.884} C_VEL
LIN {X 0,Y 237.965,Z 642.387,A -85,B 0,C 180,E1 -19638.325,E2 -19638.325} C_VEL
LIN {X 0,Y 236.445,Z 621.747,A -85,B 0,C 180,E1 -19639.366,E2 -19639.366} C_VEL
LIN {X 0,Y 236.409,Z 617.267,A -85,B 0,C 180,E1 -19639.652,E2 -19639.652} C_VEL
LIN {X 0,Y 238.156,Z 597.6,A -85,B 0,C 180,E1 -19644.402,E2 -19644.402} C_VEL
LIN {X 0,Y 239.912,Z 579.97,A -85,B 0,C 180,E1 -19648.653,E2 -19648.653} C_VEL
LIN {X 0,Y 238.389,Z 571.606,A -85,B 0,C 180,E1 -19650.794,E2 -19650.794} C_VEL
LIN {X 0,Y 235.102,Z 555.352,A -85,B 0,C 180,E1 -19655.126,E2 -19655.126} C_VEL
LIN {X 0,Y 234.946,Z 555.202,A -85,B 0,C 180,E1 -19658.944,E2 -19658.944} C_VEL
LIN {X 0,Y 234.884,Z 555.168,A -85,B 0,C 180,E1 -19663.487,E2 -19663.487} C_VEL
LIN {X 0,Y 234.889,Z 555.227,A -85,B 0,C 180,E1 -19666.513,E2 -19666.513} C_VEL
LIN {X 0,Y 234.922,Z 555.181,A -85,B 0,C 180,E1 -19671.078,E2 -19671.078} C_VEL
LIN {X 0,Y 234.982,Z 555.43,A -85,B 0,C 180,E1 -19674.023,E2 -19674.023} C_VEL
LIN {X 0,Y 235.313,Z 556.707,A -85,B 0,C 180,E1 -19674.458,E2 -19674.458} C_VEL
LIN {X 0,Y 241.781,Z 568.667,A -85,B 0,C 180,E1 -19676.009,E2 -19676.009} C_VEL
LIN {X 0,Y 249.378,Z 584.591,A -85,B 0,C 180,E1 -19677.722,E2 -19677.722} C_VEL
LIN {X 0,Y 254.994,Z 598.56,A -85,B 0,C 180,E1 -19678.975,E2 -19678.975} C_VEL
LIN {X 0,Y 253.351,Z 648.553,A -85,B 0,C 180,E1 -19680.363,E2 -19680.363} C_VEL
LIN {X 0,Y 252.481,Z 665.721,A -85,B 0,C 180,E1 -19680.898,E2 -19680.898} C_VEL
LIN {X 0,Y 251.327,Z 678.749,A -85,B 0,C 180,E1 -19681.615,E2 -19681.615} C_VEL
LIN {X 0,Y 249.853,Z 690.555,A -85,B 0,C 180,E1 -19682.573,E2 -19682.573} C_VEL
LIN {X 0,Y 247.855,Z 702.931,A -85,B 0,C 180,E1 -19683.926,E2 -19683.926} C_VEL
LIN {X 0,Y 245.716,Z 713.972,A -85,B 0,C 180,E1 -19685.496,E2 -19685.496} C_VEL
LIN {X 0,Y 243.627,Z 723.311,A -85,B 0,C 180,E1 -19687.169,E2 -19687.169} C_VEL
LIN {X 0,Y 241.653,Z 732.206,A -85,B 0,C 180,E1 -19689.165,E2 -19689.165} C_VEL
LIN {X 0,Y 239.274,Z 740.979,A -85,B 0,C 180,E1 -19691.592,E2 -19691.592} C_VEL
LIN {X 0,Y 237.309,Z 748.144,A -85,B 0,C 180,E1 -19694.1,E2 -19694.1} C_VEL
LIN {X 0,Y 235.946,Z 752.977,A -85,B 0,C 180,E1 -19696.213,E2 -19696.213} C_VEL
LIN {X 0,Y 234.646,Z 757.671,A -85,B 0,C 180,E1 -19698.772,E2 -19698.772} C_VEL
LIN {X 0,Y 233.795,Z 761.254,A -85,B 0,C 180,E1 -19701.354,E2 -19701.354} C_VEL
LIN {X 0,Y 233.226,Z 763.837,A -85,B 0,C 180,E1 -19703.945,E2 -19703.945} C_VEL
LIN {X 0,Y 232.96,Z 765.487,A -85,B 0,C 180,E1 -19706.539,E2 -19706.539} C_VEL
LIN {X 0,Y 232.835,Z 766.326,A -85,B 0,C 180,E1 -19709.999,E2 -19709.999} C_VEL
LIN {X 0,Y 232.835,Z 766.134,A -85,B 0,C 180,E1 -19711.728,E2 -19711.728} C_VEL
LIN {X 0,Y 232.958,Z 765.549,A -85,B 0,C 180,E1 -19713.458,E2 -19713.458} C_VEL
LIN {X 0,Y 233.387,Z 763.229,A -85,B 0,C 180,E1 -19716.917,E2 -19716.917} C_VEL
LIN {X 0,Y 234.03,Z 760.361,A -85,B 0,C 180,E1 -19719.505,E2 -19719.505} C_VEL
LIN {X 0,Y 235.014,Z 756.469,A -85,B 0,C 180,E1 -19722.082,E2 -19722.082} C_VEL
LIN {X 0,Y 236.406,Z 751.45,A -85,B 0,C 180,E1 -19724.635,E2 -19724.635} C_VEL
LIN {X 0,Y 238.088,Z 745.13,A -85,B 0,C 180,E1 -19727.167,E2 -19727.167} C_VEL
LIN {X 0,Y 240.36,Z 737.211,A -85,B 0,C 180,E1 -19729.647,E2 -19729.647} C_VEL
LIN {X 0,Y 242.444,Z 728.895,A -85,B 0,C 180,E1 -19731.752,E2 -19731.752} C_VEL
LIN {X 0,Y 244.592,Z 719.296,A -85,B 0,C 180,E1 -19733.718,E2 -19733.718} C_VEL
LIN {X 0,Y 246.901,Z 708.208,A -85,B 0,C 180,E1 -19735.499,E2 -19735.499} C_VEL
LIN {X 0,Y 248.955,Z 697.328,A -85,B 0,C 180,E1 -19736.85,E2 -19736.85} C_VEL
LIN {X 0,Y 250.657,Z 685.298,A -85,B 0,C 180,E1 -19738.009,E2 -19738.009} C_VEL
LIN {X 0,Y 251.986,Z 672.926,A -85,B 0,C 180,E1 -19738.87,E2 -19738.87} C_VEL
LIN {X 0,Y 252.977,Z 660.071,A -85,B 0,C 180,E1 -19739.429,E2 -19739.429} C_VEL
LIN {X 0,Y 255.097,Z 598.761,A -85,B 0,C 180,E1 -19741.138,E2 -19741.138} C_VEL
LIN {X 0,Y 249.282,Z 584.356,A -85,B 0,C 180,E1 -19742.436,E2 -19742.436} C_VEL
LIN {X 0,Y 241.15,Z 567.4,A -85,B 0,C 180,E1 -19744.279,E2 -19744.279} C_VEL
LIN {X 0,Y 235.213,Z 556.368,A -85,B 0,C 180,E1 -19745.743,E2 -19745.743} C_VEL
LIN {X 0,Y 234.974,Z 555.281,A -85,B 0,C 180,E1 -19746.267,E2 -19746.267} C_VEL
LIN {X 0,Y 234.939,Z 555.208,A -85,B 0,C 180,E1 -19748.943,E2 -19748.943} C_VEL
LIN {X 0,Y 234.884,Z 555.213,A -85,B 0,C 180,E1 -19753.484,E2 -19753.484} C_VEL
LIN {X 0,Y 234.916,Z 555.211,A -85,B 0,C 180,E1 -19756.52,E2 -19756.52} C_VEL
LIN {X 0,Y 234.95,Z 555.185,A -85,B 0,C 180,E1 -19761.085,E2 -19761.085} C_VEL
LIN {X 0,Y 234.956,Z 555.221,A -85,B 0,C 180,E1 -19765.366,E2 -19765.366} C_VEL
LIN {X 0,Y 234.964,Z 555.217,A -85,B 0,C 180,E1 -19770.156,E2 -19770.156} C_VEL
LIN {X 0,Y 234.988,Z 555.208,A -85,B 0,C 180,E1 -19773.793,E2 -19773.793} C_VEL
LIN {X 0,Y 235.005,Z 555.201,A -85,B 0,C 180,E1 -19778.969,E2 -19778.969} C_VEL
LIN {X 0,Y 235.09,Z 555.186,A -85,B 0,C 180,E1 -19783.059,E2 -19783.059} C_VEL
LIN {X 0,Y 235.14,Z 555.19,A -85,B 0,C 180,E1 -19787.923,E2 -19787.923} C_VEL
LIN {X 0,Y 235.362,Z 555.154,A -85,B 0,C 180,E1 -19791.646,E2 -19791.646} C_VEL
LIN {X 0,Y 235.217,Z 555.181,A -85,B 0,C 180,E1 -19794.857,E2 -19794.857} C_VEL
LIN {X 0,Y 235.593,Z 555.129,A -85,B 0,C 180,E1 -19799.058,E2 -19799.058} C_VEL
LIN {X 0,Y 234.906,Z 555.225,A -85,B 0,C 180,E1 -19800.482,E2 -19800.482} C_VEL
LIN {X 0,Y 231.859,Z 555.595,A -85,B 0,C 180,E1 -19802.797,E2 -19802.797} C_VEL
LIN {X 0,Y 229.318,Z 555.908,A -85,B 0,C 180,E1 -19804.688,E2 -19804.688} C_VEL
LIN {X 0,Y 228.321,Z 556.044,A -85,B 0,C 180,E1 -19806.161,E2 -19806.161} C_VEL
LIN {X 0,Y 228.293,Z 556.043,A -85,B 0,C 180,E1 -19806.66,E2 -19806.66} C_VEL
LIN {X 0,Y 228.268,Z 556.033,A -85,B 0,C 180,E1 -19809.871,E2 -19809.871} C_VEL
LIN {X 0,Y 228.059,Z 556.073,A -85,B 0,C 180,E1 -19814.272,E2 -19814.272} C_VEL
LIN {X 0,Y 227.997,Z 556.08,A -85,B 0,C 180,E1 -19817.954,E2 -19817.954} C_VEL
LIN {X 0,Y 227.924,Z 556.083,A -85,B 0,C 180,E1 -19822.33,E2 -19822.33} C_VEL
LIN {X 0,Y 227.936,Z 556.08,A -85,B 0,C 180,E1 -19826.603,E2 -19826.603} C_VEL
LIN {X 0,Y 227.891,Z 556.092,A -85,B 0,C 180,E1 -19830.292,E2 -19830.292} C_VEL
LIN {X 0,Y 227.871,Z 556.098,A -85,B 0,C 180,E1 -19833.722,E2 -19833.722} C_VEL
LIN {X 0,Y 227.86,Z 556.081,A -85,B 0,C 180,E1 -19838.088,E2 -19838.088} C_VEL
LIN {X 0,Y 227.862,Z 556.081,A -85,B 0,C 180,E1 -19842.731,E2 -19842.731} C_VEL
LIN {X 0,Y 227.914,Z 556.083,A -85,B 0,C 180,E1 -19847.737,E2 -19847.737} C_VEL
LIN {X 0,Y 227.96,Z 556.387,A -85,B 0,C 180,E1 -19848.3,E2 -19848.3} C_VEL
LIN {X 0,Y 230.002,Z 564.241,A -85,B 0,C 180,E1 -19852.331,E2 -19852.331} C_VEL
LIN {X 0,Y 230.679,Z 566.88,A -85,B 0,C 180,E1 -19853.48,E2 -19853.48} C_VEL
LIN {X 0,Y 237.19,Z 580.336,A -85,B 0,C 180,E1 -19855.169,E2 -19855.169} C_VEL
LIN {X 0,Y 244.414,Z 596.832,A -85,B 0,C 180,E1 -19856.899,E2 -19856.899} C_VEL
LIN {X 0,Y 245.573,Z 600.059,A -85,B 0,C 180,E1 -19857.183,E2 -19857.183} C_VEL
LIN {X 0,Y 248.38,Z 620.834,A -85,B 0,C 180,E1 -19858.29,E2 -19858.29} C_VEL
LIN {X 0,Y 246.186,Z 675.59,A -85,B 0,C 180,E1 -19859.852,E2 -19859.852} C_VEL
LIN {X 0,Y 244.875,Z 689.466,A -85,B 0,C 180,E1 -19860.563,E2 -19860.563} C_VEL
LIN {X 0,Y 243.118,Z 701.897,A -85,B 0,C 180,E1 -19861.514,E2 -19861.514} C_VEL
LIN {X 0,Y 241.196,Z 713,A -85,B 0,C 180,E1 -19862.684,E2 -19862.684} C_VEL
LIN {X 0,Y 238.794,Z 724.564,A -85,B 0,C 180,E1 -19864.273,E2 -19864.273} C_VEL
LIN {X 0,Y 236.316,Z 734.979,A -85,B 0,C 180,E1 -19866.098,E2 -19866.098} C_VEL
LIN {X 0,Y 234.169,Z 743.5,A -85,B 0,C 180,E1 -19867.968,E2 -19867.968} C_VEL
LIN {X 0,Y 231.807,Z 752.742,A -85,B 0,C 180,E1 -19870.52,E2 -19870.52} C_VEL
LIN {X 0,Y 229.727,Z 760.17,A -85,B 0,C 180,E1 -19873.106,E2 -19873.106} C_VEL
LIN {X 0,Y 227.979,Z 766.133,A -85,B 0,C 180,E1 -19875.724,E2 -19875.724} C_VEL
LIN {X 0,Y 226.881,Z 770.855,A -85,B 0,C 180,E1 -19878.386,E2 -19878.386} C_VEL
LIN {X 0,Y 226.139,Z 774.468,A -85,B 0,C 180,E1 -19881.062,E2 -19881.062} C_VEL
LIN {X 0,Y 225.821,Z 776.331,A -85,B 0,C 180,E1 -19882.85,E2 -19882.85} C_VEL
LIN {X 0,Y 225.58,Z 778.299,A -85,B 0,C 180,E1 -19885.54,E2 -19885.54} C_VEL
LIN {X 0,Y 225.622,Z 779.335,A -85,B 0,C 180,E1 -19888.217,E2 -19888.217} C_VEL
LIN {X 0,Y 225.688,Z 779.548,A -85,B 0,C 180,E1 -19890.002,E2 -19890.002} C_VEL
LIN {X 0,Y 225.759,Z 779.29,A -85,B 0,C 180,E1 -19892.455,E2 -19892.455} C_VEL
LIN {X 0,Y 225.843,Z 781.951,A -85,B 0,C 180,E1 -19895.358,E2 -19895.358} C_VEL
LIN {X 0,Y 226.056,Z 782.895,A -85,B 0,C 180,E1 -19897.145,E2 -19897.145} C_VEL
LIN {X 0,Y 226.49,Z 783.315,A -85,B 0,C 180,E1 -19898.927,E2 -19898.927} C_VEL
LIN {X 0,Y 227.174,Z 783.285,A -85,B 0,C 180,E1 -19900.699,E2 -19900.699} C_VEL
LIN {X 0,Y 228.124,Z 782.813,A -85,B 0,C 180,E1 -19902.455,E2 -19902.455} C_VEL
LIN {X 0,Y 229.244,Z 781.805,A -85,B 0,C 180,E1 -19904.199,E2 -19904.199} C_VEL
LIN {X 0,Y 231.301,Z 779.356,A -85,B 0,C 180,E1 -19906.779,E2 -19906.779} C_VEL
LIN {X 0,Y 234.064,Z 775.678,A -85,B 0,C 180,E1 -19909.287,E2 -19909.287} C_VEL
LIN {X 0,Y 237.29,Z 770.691,A -85,B 0,C 180,E1 -19911.731,E2 -19911.731} C_VEL
LIN {X 0,Y 240.972,Z 764.381,A -85,B 0,C 180,E1 -19914.1,E2 -19914.1} C_VEL
LIN {X 0,Y 245.023,Z 756.215,A -85,B 0,C 180,E1 -19916.398,E2 -19916.398} C_VEL
LIN {X 0,Y 248.901,Z 747.771,A -85,B 0,C 180,E1 -19918.228,E2 -19918.228} C_VEL
LIN {X 0,Y 253.025,Z 737.265,A -85,B 0,C 180,E1 -19919.999,E2 -19919.999} C_VEL
LIN {X 0,Y 256.544,Z 726.713,A -85,B 0,C 180,E1 -19921.367,E2 -19921.367} C_VEL
LIN {X 0,Y 259.733,Z 715.427,A -85,B 0,C 180,E1 -19922.477,E2 -19922.477} C_VEL
LIN {X 0,Y 262.041,Z 704.461,A -85,B 0,C 180,E1 -19923.303,E2 -19923.303} C_VEL
LIN {X 0,Y 267.731,Z 672.772,A -85,B 0,C 180,E1 -19925.018,E2 -19925.018} C_VEL
LIN {X 0,Y 275.412,Z 632.018,A -85,B 0,C 180,E1 -19927.035,E2 -19927.035} C_VEL
LIN {X 0,Y 273.333,Z 629.635,A -85,B 0,C 180,E1 -19929.107,E2 -19929.107} C_VEL
LIN {X 0,Y 271.675,Z 628.281,A -85,B 0,C 180,E1 -19931.392,E2 -19931.392} C_VEL
LIN {X 0,Y 270.561,Z 628.156,A -85,B 0,C 180,E1 -19934.089,E2 -19934.089} C_VEL
LIN {X 0,Y 270.387,Z 629.675,A -85,B 0,C 180,E1 -19936.703,E2 -19936.703} C_VEL
LIN {X 0,Y 270.771,Z 631.573,A -85,B 0,C 180,E1 -19938.549,E2 -19938.549} C_VEL
LIN {X 0,Y 271.911,Z 636.411,A -85,B 0,C 180,E1 -19941.188,E2 -19941.188} C_VEL
LIN {X 0,Y 272.274,Z 639.048,A -85,B 0,C 180,E1 -19942.062,E2 -19942.062} C_VEL
LIN {X 0,Y 272.093,Z 651.902,A -85,B 0,C 180,E1 -19944.191,E2 -19944.191} C_VEL
LIN {X 0,Y 271.932,Z 663.542,A -85,B 0,C 180,E1 -19945.761,E2 -19945.761} C_VEL
LIN {X 0,Y 271.759,Z 665.376,A -85,B 0,C 180,E1 -19945.923,E2 -19945.923} C_VEL
LIN {X 0,Y 265.04,Z 703.889,A -85,B 0,C 180,E1 -19947.86,E2 -19947.86} C_VEL
LIN {X 0,Y 262.157,Z 715.959,A -85,B 0,C 180,E1 -19948.707,E2 -19948.707} C_VEL
LIN {X 0,Y 259.156,Z 725.795,A -85,B 0,C 180,E1 -19949.663,E2 -19949.663} C_VEL
LIN {X 0,Y 255.884,Z 735.234,A -85,B 0,C 180,E1 -19950.823,E2 -19950.823} C_VEL
LIN {X 0,Y 252.295,Z 744.082,A -85,B 0,C 180,E1 -19952.187,E2 -19952.187} C_VEL
LIN {X 0,Y 248.09,Z 752.855,A -85,B 0,C 180,E1 -19953.954,E2 -19953.954} C_VEL
LIN {X 0,Y 244.254,Z 760.085,A -85,B 0,C 180,E1 -19955.794,E2 -19955.794} C_VEL
LIN {X 0,Y 240.791,Z 765.923,A -85,B 0,C 180,E1 -19957.701,E2 -19957.701} C_VEL
LIN {X 0,Y 237.092,Z 771.406,A -85,B 0,C 180,E1 -19960.069,E2 -19960.069} C_VEL
LIN {X 0,Y 234.936,Z 774.32,A -85,B 0,C 180,E1 -19961.693,E2 -19961.693} C_VEL
LIN {X 0,Y 232.023,Z 777.515,A -85,B 0,C 180,E1 -19964.18,E2 -19964.18} C_VEL
LIN {X 0,Y 230.413,Z 779.05,A -85,B 0,C 180,E1 -19965.876,E2 -19965.876} C_VEL
LIN {X 0,Y 229.08,Z 780.009,A -85,B 0,C 180,E1 -19967.599,E2 -19967.599} C_VEL
LIN {X 0,Y 227.995,Z 780.454,A -85,B 0,C 180,E1 -19969.342,E2 -19969.342} C_VEL
LIN {X 0,Y 227.177,Z 780.446,A -85,B 0,C 180,E1 -19971.102,E2 -19971.102} C_VEL
LIN {X 0,Y 226.359,Z 779.637,A -85,B 0,C 180,E1 -19973.491,E2 -19973.491} C_VEL
LIN {X 0,Y 226.063,Z 778.971,A -85,B 0,C 180,E1 -19974.649,E2 -19974.649} C_VEL
LIN {X 0,Y 225.8,Z 776.462,A -85,B 0,C 180,E1 -19977.324,E2 -19977.324} C_VEL
LIN {X 0,Y 225.785,Z 772.641,A -85,B 0,C 180,E1 -19980,E2 -19980} C_VEL
LIN {X 0,Y 226.008,Z 767.441,A -85,B 0,C 180,E1 -19982.674,E2 -19982.674} C_VEL
LIN {X 0,Y 226.222,Z 761.785,A -85,B 0,C 180,E1 -19984.901,E2 -19984.901} C_VEL
LIN {X 0,Y 226.604,Z 754.591,A -85,B 0,C 180,E1 -19987.126,E2 -19987.126} C_VEL
LIN {X 0,Y 226.934,Z 747.49,A -85,B 0,C 180,E1 -19988.908,E2 -19988.908} C_VEL
LIN {X 0,Y 227.451,Z 738.913,A -85,B 0,C 180,E1 -19990.684,E2 -19990.684} C_VEL
LIN {X 0,Y 228.108,Z 728.17,A -85,B 0,C 180,E1 -19992.455,E2 -19992.455} C_VEL
LIN {X 0,Y 228.743,Z 717.738,A -85,B 0,C 180,E1 -19993.775,E2 -19993.775} C_VEL
LIN {X 0,Y 229.216,Z 706.375,A -85,B 0,C 180,E1 -19994.88,E2 -19994.88} C_VEL
LIN {X 0,Y 229.647,Z 693.742,A -85,B 0,C 180,E1 -19995.703,E2 -19995.703} C_VEL
LIN {X 0,Y 230.975,Z 644.063,A -85,B 0,C 180,E1 -19998.294,E2 -19998.294} C_VEL
LIN {X 0,Y 229.364,Z 621.171,A -85,B 0,C 180,E1 -19999.504,E2 -19999.504} C_VEL
LIN {X 0,Y 229.338,Z 617.294,A -85,B 0,C 180,E1 -19999.758,E2 -19999.758} C_VEL
LIN {X 0,Y 231.206,Z 596.755,A -85,B 0,C 180,E1 -20004.839,E2 -20004.839} C_VEL
LIN {X 0,Y 232.856,Z 580.391,A -85,B 0,C 180,E1 -20008.876,E2 -20008.876} C_VEL
LIN {X 0,Y 229.827,Z 565.116,A -85,B 0,C 180,E1 -20012.906,E2 -20012.906} C_VEL
LIN {X 0,Y 228.048,Z 556.245,A -85,B 0,C 180,E1 -20015.365,E2 -20015.365} C_VEL
LIN {X 0,Y 227.836,Z 556.053,A -85,B 0,C 180,E1 -20020.375,E2 -20020.375} C_VEL
LIN {X 0,Y 227.834,Z 556.076,A -85,B 0,C 180,E1 -20025.193,E2 -20025.193} C_VEL
LIN {X 0,Y 227.816,Z 556.064,A -85,B 0,C 180,E1 -20029.62,E2 -20029.62} C_VEL
LIN {X 0,Y 227.888,Z 556.224,A -85,B 0,C 180,E1 -20032.783,E2 -20032.783} C_VEL
LIN {X 0,Y 228.134,Z 557.235,A -85,B 0,C 180,E1 -20033.174,E2 -20033.174} C_VEL
LIN {X 0,Y 229.694,Z 559.998,A -85,B 0,C 180,E1 -20033.603,E2 -20033.603} C_VEL
LIN {X 0,Y 234.887,Z 569.155,A -85,B 0,C 180,E1 -20034.876,E2 -20034.876} C_VEL
LIN {X 0,Y 242.032,Z 583.806,A -85,B 0,C 180,E1 -20036.58,E2 -20036.58} C_VEL
LIN {X 0,Y 247.61,Z 597.031,A -85,B 0,C 180,E1 -20037.881,E2 -20037.881} C_VEL
LIN {X 0,Y 248.96,Z 600.451,A -85,B 0,C 180,E1 -20038.191,E2 -20038.191} C_VEL
LIN {X 0,Y 246.52,Z 663.369,A -85,B 0,C 180,E1 -20039.991,E2 -20039.991} C_VEL
LIN {X 0,Y 245.341,Z 676.912,A -85,B 0,C 180,E1 -20040.695,E2 -20040.695} C_VEL
LIN {X 0,Y 243.715,Z 689.772,A -85,B 0,C 180,E1 -20041.704,E2 -20041.704} C_VEL
LIN {X 0,Y 241.797,Z 701.563,A -85,B 0,C 180,E1 -20042.988,E2 -20042.988} C_VEL
LIN {X 0,Y 239.556,Z 712.902,A -85,B 0,C 180,E1 -20044.591,E2 -20044.591} C_VEL
LIN {X 0,Y 237.108,Z 723.518,A -85,B 0,C 180,E1 -20046.504,E2 -20046.504} C_VEL
LIN {X 0,Y 234.981,Z 732.551,A -85,B 0,C 180,E1 -20048.583,E2 -20048.583} C_VEL
LIN {X 0,Y 232.558,Z 741.185,A -85,B 0,C 180,E1 -20051.041,E2 -20051.041} C_VEL
LIN {X 0,Y 230.474,Z 748.351,A -85,B 0,C 180,E1 -20053.615,E2 -20053.615} C_VEL
LIN {X 0,Y 229.049,Z 753.183,A -85,B 0,C 180,E1 -20055.789,E2 -20055.789} C_VEL
LIN {X 0,Y 227.692,Z 757.876,A -85,B 0,C 180,E1 -20058.425,E2 -20058.425} C_VEL
LIN {X 0,Y 226.769,Z 761.46,A -85,B 0,C 180,E1 -20061.084,E2 -20061.084} C_VEL
LIN {X 0,Y 226.109,Z 764.293,A -85,B 0,C 180,E1 -20064.066,E2 -20064.066} C_VEL
LIN {X 0,Y 225.868,Z 765.693,A -85,B 0,C 180,E1 -20066.431,E2 -20066.431} C_VEL
LIN {X 0,Y 225.748,Z 766.531,A -85,B 0,C 180,E1 -20069.998,E2 -20069.998} C_VEL
LIN {X 0,Y 225.753,Z 766.338,A -85,B 0,C 180,E1 -20071.782,E2 -20071.782} C_VEL
LIN {X 0,Y 225.865,Z 765.754,A -85,B 0,C 180,E1 -20073.566,E2 -20073.566} C_VEL
LIN {X 0,Y 226.332,Z 763.434,A -85,B 0,C 180,E1 -20077.133,E2 -20077.133} C_VEL
LIN {X 0,Y 227.023,Z 760.565,A -85,B 0,C 180,E1 -20079.802,E2 -20079.802} C_VEL
LIN {X 0,Y 228.08,Z 756.672,A -85,B 0,C 180,E1 -20082.455,E2 -20082.455} C_VEL
LIN {X 0,Y 229.54,Z 751.654,A -85,B 0,C 180,E1 -20085.083,E2 -20085.083} C_VEL
LIN {X 0,Y 231.317,Z 745.333,A -85,B 0,C 180,E1 -20087.686,E2 -20087.686} C_VEL
LIN {X 0,Y 233.696,Z 737.413,A -85,B 0,C 180,E1 -20090.231,E2 -20090.231} C_VEL
LIN {X 0,Y 235.716,Z 729.67,A -85,B 0,C 180,E1 -20092.257,E2 -20092.257} C_VEL
LIN {X 0,Y 238.1,Z 719.497,A -85,B 0,C 180,E1 -20094.407,E2 -20094.407} C_VEL
LIN {X 0,Y 240.521,Z 708.408,A -85,B 0,C 180,E1 -20096.227,E2 -20096.227} C_VEL
LIN {X 0,Y 242.655,Z 697.526,A -85,B 0,C 180,E1 -20097.605,E2 -20097.605} C_VEL
LIN {X 0,Y 244.423,Z 685.495,A -85,B 0,C 180,E1 -20098.789,E2 -20098.789} C_VEL
LIN {X 0,Y 245.877,Z 672.424,A -85,B 0,C 180,E1 -20099.703,E2 -20099.703} C_VEL
LIN {X 0,Y 246.874,Z 659.484,A -85,B 0,C 180,E1 -20100.262,E2 -20100.262} C_VEL
LIN {X 0,Y 248.982,Z 601.786,A -85,B 0,C 180,E1 -20101.897,E2 -20101.897} C_VEL
LIN {X 0,Y 248.66,Z 599.67,A -85,B 0,C 180,E1 -20102.015,E2 -20102.015} C_VEL
LIN {X 0,Y 243.031,Z 586.016,A -85,B 0,C 180,E1 -20103.327,E2 -20103.327} C_VEL
LIN {X 0,Y 235.849,Z 571.017,A -85,B 0,C 180,E1 -20105.036,E2 -20105.036} C_VEL
LIN {X 0,Y 229.88,Z 560.164,A -85,B 0,C 180,E1 -20106.506,E2 -20106.506} C_VEL
LIN {X 0,Y 228.41,Z 558.012,A -85,B 0,C 180,E1 -20106.869,E2 -20106.869} C_VEL
LIN {X 0,Y 227.89,Z 556.226,A -85,B 0,C 180,E1 -20107.183,E2 -20107.183} C_VEL
LIN {X 0,Y 227.83,Z 556.091,A -85,B 0,C 180,E1 -20110.373,E2 -20110.373} C_VEL
LIN {X 0,Y 227.832,Z 556.082,A -85,B 0,C 180,E1 -20115.191,E2 -20115.191} C_VEL
LIN {X 0,Y 227.869,Z 556.08,A -85,B 0,C 180,E1 -20119.632,E2 -20119.632} C_VEL
LIN {X 0,Y 227.897,Z 556.09,A -85,B 0,C 180,E1 -20124.131,E2 -20124.131} C_VEL
LIN {X 0,Y 227.868,Z 556.094,A -85,B 0,C 180,E1 -20128.377,E2 -20128.377} C_VEL
LIN {X 0,Y 227.88,Z 556.085,A -85,B 0,C 180,E1 -20132.444,E2 -20132.444} C_VEL
LIN {X 0,Y 227.908,Z 556.09,A -85,B 0,C 180,E1 -20136.367,E2 -20136.367} C_VEL
LIN {X 0,Y 227.937,Z 556.091,A -85,B 0,C 180,E1 -20140.174,E2 -20140.174} C_VEL
LIN {X 0,Y 228.051,Z 556.06,A -85,B 0,C 180,E1 -20143.897,E2 -20143.897} C_VEL
LIN {X 0,Y 228.088,Z 556.071,A -85,B 0,C 180,E1 -20147.544,E2 -20147.544} C_VEL
LIN {X 0,Y 228.3,Z 556.031,A -85,B 0,C 180,E1 -20151.146,E2 -20151.146} C_VEL
LIN {X 0,Y 228.349,Z 556.039,A -85,B 0,C 180,E1 -20152.928,E2 -20152.928} C_VEL
LIN {X 0,Y 228.555,Z 556.005,A -85,B 0,C 180,E1 -20159.073,E2 -20159.073} C_VEL
LIN {X 0,Y 228.549,Z 556.009,A -85,B 0,C 180,E1 -20161.762,E2 -20161.762} C_VEL
LIN {X 0,Y 228.293,Z 556.043,A -85,B 0,C 180,E1 -20166.66,E2 -20166.66} C_VEL
LIN {X 0,Y 227.72,Z 556.123,A -85,B 0,C 180,E1 -20168.131,E2 -20168.131} C_VEL
LIN {X 0,Y 226.097,Z 556.326,A -85,B 0,C 180,E1 -20169.572,E2 -20169.572} C_VEL
LIN {X 0,Y 222.151,Z 556.811,A -85,B 0,C 180,E1 -20172.478,E2 -20172.478} C_VEL
LIN {X 0,Y 221.055,Z 556.946,A -85,B 0,C 180,E1 -20174.002,E2 -20174.002} C_VEL
LIN {X 0,Y 220.981,Z 556.95,A -85,B 0,C 180,E1 -20174.52,E2 -20174.52} C_VEL
LIN {X 0,Y 220.978,Z 556.949,A -85,B 0,C 180,E1 -20177.429,E2 -20177.429} C_VEL
LIN {X 0,Y 220.89,Z 556.961,A -85,B 0,C 180,E1 -20182.683,E2 -20182.683} C_VEL
LIN {X 0,Y 220.877,Z 556.96,A -85,B 0,C 180,E1 -20187.015,E2 -20187.015} C_VEL
LIN {X 0,Y 220.833,Z 556.969,A -85,B 0,C 180,E1 -20190.769,E2 -20190.769} C_VEL
LIN {X 0,Y 220.795,Z 556.961,A -85,B 0,C 180,E1 -20194.956,E2 -20194.956} C_VEL
LIN {X 0,Y 220.829,Z 556.978,A -85,B 0,C 180,E1 -20199.532,E2 -20199.532} C_VEL
LIN {X 0,Y 220.811,Z 556.974,A -85,B 0,C 180,E1 -20204.445,E2 -20204.445} C_VEL
LIN {X 0,Y 220.869,Z 557.068,A -85,B 0,C 180,E1 -20207.042,E2 -20207.042} C_VEL
LIN {X 0,Y 222.874,Z 564.567,A -85,B 0,C 180,E1 -20211.174,E2 -20211.174} C_VEL
LIN {X 0,Y 223.4,Z 566.7,A -85,B 0,C 180,E1 -20212.093,E2 -20212.093} C_VEL
LIN {X 0,Y 230.121,Z 580.026,A -85,B 0,C 180,E1 -20213.931,E2 -20213.931} C_VEL
LIN {X 0,Y 237.565,Z 596.705,A -85,B 0,C 180,E1 -20215.818,E2 -20215.818} C_VEL
LIN {X 0,Y 239.801,Z 602.53,A -85,B 0,C 180,E1 -20216.383,E2 -20216.383} C_VEL
LIN {X 0,Y 242.323,Z 621.674,A -85,B 0,C 180,E1 -20217.436,E2 -20217.436} C_VEL
LIN {X 0,Y 240.045,Z 675.898,A -85,B 0,C 180,E1 -20219.024,E2 -20219.024} C_VEL
LIN {X 0,Y 238.721,Z 689.342,A -85,B 0,C 180,E1 -20219.732,E2 -20219.732} C_VEL
LIN {X 0,Y 236.902,Z 701.699,A -85,B 0,C 180,E1 -20220.695,E2 -20220.695} C_VEL
LIN {X 0,Y 234.914,Z 712.801,A -85,B 0,C 180,E1 -20221.89,E2 -20221.89} C_VEL
LIN {X 0,Y 232.413,Z 724.363,A -85,B 0,C 180,E1 -20223.513,E2 -20223.513} C_VEL
LIN {X 0,Y 229.845,Z 734.777,A -85,B 0,C 180,E1 -20225.381,E2 -20225.381} C_VEL
LIN {X 0,Y 227.563,Z 743.297,A -85,B 0,C 180,E1 -20227.293,E2 -20227.293} C_VEL
LIN {X 0,Y 225.599,Z 750.738,A -85,B 0,C 180,E1 -20229.349,E2 -20229.349} C_VEL
LIN {X 0,Y 223.187,Z 758.843,A -85,B 0,C 180,E1 -20232.122,E2 -20232.122} C_VEL
LIN {X 0,Y 221.084,Z 765.93,A -85,B 0,C 180,E1 -20235.269,E2 -20235.269} C_VEL
LIN {X 0,Y 219.887,Z 770.65,A -85,B 0,C 180,E1 -20238.011,E2 -20238.011} C_VEL
LIN {X 0,Y 219.091,Z 774.263,A -85,B 0,C 180,E1 -20240.772,E2 -20240.772} C_VEL
LIN {X 0,Y 218.759,Z 776.126,A -85,B 0,C 180,E1 -20242.618,E2 -20242.618} C_VEL
LIN {X 0,Y 218.481,Z 778.255,A -85,B 0,C 180,E1 -20245.71,E2 -20245.71} C_VEL
LIN {X 0,Y 218.522,Z 779.13,A -85,B 0,C 180,E1 -20248.159,E2 -20248.159} C_VEL
LIN {X 0,Y 218.604,Z 779.344,A -85,B 0,C 180,E1 -20250.002,E2 -20250.002} C_VEL
LIN {X 0,Y 218.721,Z 778.919,A -85,B 0,C 180,E1 -20252.995,E2 -20252.995} C_VEL
LIN {X 0,Y 218.797,Z 781.309,A -85,B 0,C 180,E1 -20255.531,E2 -20255.531} C_VEL
LIN {X 0,Y 219.02,Z 782.442,A -85,B 0,C 180,E1 -20257.376,E2 -20257.376} C_VEL
LIN {X 0,Y 219.476,Z 783.115,A -85,B 0,C 180,E1 -20259.215,E2 -20259.215} C_VEL
LIN {X 0,Y 220.207,Z 783.345,A -85,B 0,C 180,E1 -20261.041,E2 -20261.041} C_VEL
LIN {X 0,Y 221.189,Z 782.999,A -85,B 0,C 180,E1 -20262.852,E2 -20262.852} C_VEL
LIN {X 0,Y 222.365,Z 782.169,A -85,B 0,C 180,E1 -20264.647,E2 -20264.647} C_VEL
LIN {X 0,Y 223.777,Z 780.915,A -85,B 0,C 180,E1 -20266.42,E2 -20266.42} C_VEL
LIN {X 0,Y 225.449,Z 779.198,A -85,B 0,C 180,E1 -20268.165,E2 -20268.165} C_VEL
LIN {X 0,Y 228.584,Z 775.477,A -85,B 0,C 180,E1 -20270.708,E2 -20270.708} C_VEL
LIN {X 0,Y 232.136,Z 770.553,A -85,B 0,C 180,E1 -20273.179,E2 -20273.179} C_VEL
LIN {X 0,Y 235.431,Z 765.343,A -85,B 0,C 180,E1 -20275.177,E2 -20275.177} C_VEL
LIN {X 0,Y 239.846,Z 757.706,A -85,B 0,C 180,E1 -20277.486,E2 -20277.486} C_VEL
LIN {X 0,Y 243.936,Z 749.534,A -85,B 0,C 180,E1 -20279.328,E2 -20279.328} C_VEL
LIN {X 0,Y 247.898,Z 740.763,A -85,B 0,C 180,E1 -20280.922,E2 -20280.922} C_VEL
LIN {X 0,Y 252.064,Z 729.826,A -85,B 0,C 180,E1 -20282.462,E2 -20282.462} C_VEL
LIN {X 0,Y 255.779,Z 718.206,A -85,B 0,C 180,E1 -20283.691,E2 -20283.691} C_VEL
LIN {X 0,Y 258.864,Z 705.811,A -85,B 0,C 180,E1 -20284.665,E2 -20284.665} C_VEL
LIN {X 0,Y 262.357,Z 687.387,A -85,B 0,C 180,E1 -20285.711,E2 -20285.711} C_VEL
LIN {X 0,Y 272.276,Z 637.544,A -85,B 0,C 180,E1 -20288.204,E2 -20288.204} C_VEL
LIN {X 0,Y 270.418,Z 635.525,A -85,B 0,C 180,E1 -20290.523,E2 -20290.523} C_VEL
LIN {X 0,Y 269.127,Z 634.954,A -85,B 0,C 180,E1 -20293.013,E2 -20293.013} C_VEL
LIN {X 0,Y 268.625,Z 635.579,A -85,B 0,C 180,E1 -20295.308,E2 -20295.308} C_VEL
LIN {X 0,Y 268.809,Z 637.952,A -85,B 0,C 180,E1 -20298.029,E2 -20298.029} C_VEL
LIN {X 0,Y 269.632,Z 642.5,A -85,B 0,C 180,E1 -20300.585,E2 -20300.585} C_VEL
LIN {X 0,Y 269.802,Z 644.052,A -85,B 0,C 180,E1 -20301.103,E2 -20301.103} C_VEL
LIN {X 0,Y 269.289,Z 655.454,A -85,B 0,C 180,E1 -20303.037,E2 -20303.037} C_VEL
LIN {X 0,Y 268.739,Z 666.7,A -85,B 0,C 180,E1 -20304.587,E2 -20304.587} C_VEL
LIN {X 0,Y 261.907,Z 703.522,A -85,B 0,C 180,E1 -20306.454,E2 -20306.454} C_VEL
LIN {X 0,Y 259.26,Z 714.088,A -85,B 0,C 180,E1 -20307.169,E2 -20307.169} C_VEL
LIN {X 0,Y 255.538,Z 725.963,A -85,B 0,C 180,E1 -20308.265,E2 -20308.265} C_VEL
LIN {X 0,Y 251.577,Z 736.487,A -85,B 0,C 180,E1 -20309.58,E2 -20309.58} C_VEL
LIN {X 0,Y 247.307,Z 745.887,A -85,B 0,C 180,E1 -20311.111,E2 -20311.111} C_VEL
LIN {X 0,Y 243.755,Z 752.847,A -85,B 0,C 180,E1 -20312.528,E2 -20312.528} C_VEL
LIN {X 0,Y 239.617,Z 760.006,A -85,B 0,C 180,E1 -20314.366,E2 -20314.366} C_VEL
LIN {X 0,Y 235.836,Z 765.85,A -85,B 0,C 180,E1 -20316.278,E2 -20316.278} C_VEL
LIN {X 0,Y 231.792,Z 771.373,A -85,B 0,C 180,E1 -20318.664,E2 -20318.664} C_VEL
LIN {X 0,Y 228.303,Z 775.41,A -85,B 0,C 180,E1 -20321.142,E2 -20321.142} C_VEL
LIN {X 0,Y 225.243,Z 778.3,A -85,B 0,C 180,E1 -20323.691,E2 -20323.691} C_VEL
LIN {X 0,Y 223.572,Z 779.562,A -85,B 0,C 180,E1 -20325.435,E2 -20325.435} C_VEL
LIN {X 0,Y 222.162,Z 780.367,A -85,B 0,C 180,E1 -20327.206,E2 -20327.206} C_VEL
LIN {X 0,Y 221.041,Z 780.648,A -85,B 0,C 180,E1 -20329.002,E2 -20329.002} C_VEL
LIN {X 0,Y 220.163,Z 780.374,A -85,B 0,C 180,E1 -20330.816,E2 -20330.816} C_VEL
LIN {X 0,Y 219.256,Z 779.148,A -85,B 0,C 180,E1 -20333.559,E2 -20333.559} C_VEL
LIN {X 0,Y 218.824,Z 776.793,A -85,B 0,C 180,E1 -20336.317,E2 -20336.317} C_VEL
LIN {X 0,Y 218.741,Z 773.085,A -85,B 0,C 180,E1 -20339.08,E2 -20339.08} C_VEL
LIN {X 0,Y 218.909,Z 768.002,A -85,B 0,C 180,E1 -20341.84,E2 -20341.84} C_VEL
LIN {X 0,Y 219.154,Z 762.547,A -85,B 0,C 180,E1 -20344.138,E2 -20344.138} C_VEL
LIN {X 0,Y 219.531,Z 754.634,A -85,B 0,C 180,E1 -20346.737,E2 -20346.737} C_VEL
LIN {X 0,Y 219.892,Z 746.853,A -85,B 0,C 180,E1 -20348.732,E2 -20348.732} C_VEL
LIN {X 0,Y 220.487,Z 736.979,A -85,B 0,C 180,E1 -20350.793,E2 -20350.793} C_VEL
LIN {X 0,Y 221.107,Z 727.115,A -85,B 0,C 180,E1 -20352.389,E2 -20352.389} C_VEL
LIN {X 0,Y 221.635,Z 718.413,A -85,B 0,C 180,E1 -20353.525,E2 -20353.525} C_VEL
LIN {X 0,Y 222.125,Z 707.293,A -85,B 0,C 180,E1 -20354.662,E2 -20354.662} C_VEL
LIN {X 0,Y 222.519,Z 694.397,A -85,B 0,C 180,E1 -20355.573,E2 -20355.573} C_VEL
LIN {X 0,Y 223.94,Z 645.159,A -85,B 0,C 180,E1 -20358.291,E2 -20358.291} C_VEL
LIN {X 0,Y 222.297,Z 621.39,A -85,B 0,C 180,E1 -20359.585,E2 -20359.585} C_VEL
LIN {X 0,Y 222.252,Z 617.409,A -85,B 0,C 180,E1 -20359.844,E2 -20359.844} C_VEL
LIN {X 0,Y 224.161,Z 596.819,A -85,B 0,C 180,E1 -20365.05,E2 -20365.05} C_VEL
LIN {X 0,Y 225.76,Z 582.074,A -85,B 0,C 180,E1 -20368.77,E2 -20368.77} C_VEL
LIN {X 0,Y 225.138,Z 577.547,A -85,B 0,C 180,E1 -20369.965,E2 -20369.965} C_VEL
LIN {X 0,Y 221.478,Z 559.675,A -85,B 0,C 180,E1 -20374.833,E2 -20374.833} C_VEL
LIN {X 0,Y 220.993,Z 557.088,A -85,B 0,C 180,E1 -20375.653,E2 -20375.653} C_VEL
LIN {X 0,Y 220.804,Z 556.931,A -85,B 0,C 180,E1 -20380.189,E2 -20380.189} C_VEL
LIN {X 0,Y 220.774,Z 556.937,A -85,B 0,C 180,E1 -20384.454,E2 -20384.454} C_VEL
LIN {X 0,Y 220.769,Z 556.96,A -85,B 0,C 180,E1 -20388.046,E2 -20388.046} C_VEL
LIN {X 0,Y 220.817,Z 557.074,A -85,B 0,C 180,E1 -20391.362,E2 -20391.362} C_VEL
LIN {X 0,Y 221.042,Z 558.02,A -85,B 0,C 180,E1 -20391.798,E2 -20391.798} C_VEL
LIN {X 0,Y 222.507,Z 560.744,A -85,B 0,C 180,E1 -20392.245,E2 -20392.245} C_VEL
LIN {X 0,Y 223.908,Z 562.89,A -85,B 0,C 180,E1 -20392.609,E2 -20392.609} C_VEL
LIN {X 0,Y 227.64,Z 568.98,A -85,B 0,C 180,E1 -20393.564,E2 -20393.564} C_VEL
LIN {X 0,Y 235.657,Z 585,A -85,B 0,C 180,E1 -20395.585,E2 -20395.585} C_VEL
LIN {X 0,Y 241.212,Z 598.075,A -85,B 0,C 180,E1 -20396.949,E2 -20396.949} C_VEL
LIN {X 0,Y 242.845,Z 602.195,A -85,B 0,C 180,E1 -20397.344,E2 -20397.344} C_VEL
LIN {X 0,Y 240.441,Z 663.23,A -85,B 0,C 180,E1 -20399.132,E2 -20399.132} C_VEL
LIN {X 0,Y 239.245,Z 676.523,A -85,B 0,C 180,E1 -20399.824,E2 -20399.824} C_VEL
LIN {X 0,Y 237.707,Z 688.895,A -85,B 0,C 180,E1 -20400.8,E2 -20400.8} C_VEL
LIN {X 0,Y 235.804,Z 700.191,A -85,B 0,C 180,E1 -20402.002,E2 -20402.002} C_VEL
LIN {X 0,Y 233.422,Z 711.824,A -85,B 0,C 180,E1 -20403.633,E2 -20403.633} C_VEL
LIN {X 0,Y 230.957,Z 722.271,A -85,B 0,C 180,E1 -20405.504,E2 -20405.504} C_VEL
LIN {X 0,Y 228.721,Z 731.612,A -85,B 0,C 180,E1 -20407.633,E2 -20407.633} C_VEL
LIN {X 0,Y 226.249,Z 740.045,A -85,B 0,C 180,E1 -20410.018,E2 -20410.018} C_VEL
LIN {X 0,Y 223.971,Z 747.449,A -85,B 0,C 180,E1 -20412.655,E2 -20412.655} C_VEL
LIN {X 0,Y 222.172,Z 753.39,A -85,B 0,C 180,E1 -20415.34,E2 -20415.34} C_VEL
LIN {X 0,Y 220.725,Z 758.083,A -85,B 0,C 180,E1 -20418.054,E2 -20418.054} C_VEL
LIN {X 0,Y 219.767,Z 761.665,A -85,B 0,C 180,E1 -20420.798,E2 -20420.798} C_VEL
LIN {X 0,Y 219.001,Z 764.723,A -85,B 0,C 180,E1 -20424.173,E2 -20424.173} C_VEL
LIN {X 0,Y 218.779,Z 765.898,A -85,B 0,C 180,E1 -20426.315,E2 -20426.315} C_VEL
LIN {X 0,Y 218.674,Z 766.507,A -85,B 0,C 180,E1 -20428.157,E2 -20428.157} C_VEL
LIN {X 0,Y 218.663,Z 766.735,A -85,B 0,C 180,E1 -20429.998,E2 -20429.998} C_VEL
LIN {X 0,Y 218.673,Z 766.542,A -85,B 0,C 180,E1 -20431.84,E2 -20431.84} C_VEL
LIN {X 0,Y 218.776,Z 765.958,A -85,B 0,C 180,E1 -20433.682,E2 -20433.682} C_VEL
LIN {X 0,Y 219,Z 764.813,A -85,B 0,C 180,E1 -20435.824,E2 -20435.824} C_VEL
LIN {X 0,Y 219.765,Z 761.824,A -85,B 0,C 180,E1 -20439.199,E2 -20439.199} C_VEL
LIN {X 0,Y 220.709,Z 758.291,A -85,B 0,C 180,E1 -20441.944,E2 -20441.944} C_VEL
LIN {X 0,Y 222.125,Z 753.655,A -85,B 0,C 180,E1 -20444.66,E2 -20444.66} C_VEL
LIN {X 0,Y 224.205,Z 746.669,A -85,B 0,C 180,E1 -20447.794,E2 -20447.794} C_VEL
LIN {X 0,Y 226.611,Z 739.086,A -85,B 0,C 180,E1 -20450.418,E2 -20450.418} C_VEL
LIN {X 0,Y 228.985,Z 730.513,A -85,B 0,C 180,E1 -20452.775,E2 -20452.775} C_VEL
LIN {X 0,Y 231.401,Z 720.764,A -85,B 0,C 180,E1 -20454.921,E2 -20454.921} C_VEL
LIN {X 0,Y 233.91,Z 710.001,A -85,B 0,C 180,E1 -20456.786,E2 -20456.786} C_VEL
LIN {X 0,Y 236.06,Z 699.489,A -85,B 0,C 180,E1 -20458.203,E2 -20458.203} C_VEL
LIN {X 0,Y 237.924,Z 687.947,A -85,B 0,C 180,E1 -20459.41,E2 -20459.41} C_VEL
LIN {X 0,Y 239.56,Z 674.489,A -85,B 0,C 180,E1 -20460.432,E2 -20460.432} C_VEL
LIN {X 0,Y 240.628,Z 662.185,A -85,B 0,C 180,E1 -20461.031,E2 -20461.031} C_VEL
LIN {X 0,Y 242.963,Z 602.402,A -85,B 0,C 180,E1 -20462.77,E2 -20462.77} C_VEL
LIN {X 0,Y 237.591,Z 589.344,A -85,B 0,C 180,E1 -20464.08,E2 -20464.08} C_VEL
LIN {X 0,Y 230.223,Z 573.851,A -85,B 0,C 180,E1 -20465.923,E2 -20465.923} C_VEL
LIN {X 0,Y 225.104,Z 564.735,A -85,B 0,C 180,E1 -20467.237,E2 -20467.237} C_VEL
LIN {X 0,Y 222.775,Z 561.034,A -85,B 0,C 180,E1 -20467.845,E2 -20467.845} C_VEL
LIN {X 0,Y 221.227,Z 558.587,A -85,B 0,C 180,E1 -20468.258,E2 -20468.258} C_VEL
LIN {X 0,Y 220.816,Z 556.984,A -85,B 0,C 180,E1 -20468.5,E2 -20468.5} C_VEL
LIN {X 0,Y 220.766,Z 556.978,A -85,B 0,C 180,E1 -20472.929,E2 -20472.929} C_VEL
LIN {X 0,Y 220.805,Z 556.975,A -85,B 0,C 180,E1 -20477.057,E2 -20477.057} C_VEL
LIN {X 0,Y 220.846,Z 556.944,A -85,B 0,C 180,E1 -20480.471,E2 -20480.471} C_VEL
LIN {X 0,Y 220.811,Z 556.981,A -85,B 0,C 180,E1 -20485.047,E2 -20485.047} C_VEL
LIN {X 0,Y 220.863,Z 556.973,A -85,B 0,C 180,E1 -20489.394,E2 -20489.394} C_VEL
LIN {X 0,Y 220.89,Z 556.961,A -85,B 0,C 180,E1 -20493.549,E2 -20493.549} C_VEL
LIN {X 0,Y 220.872,Z 556.956,A -85,B 0,C 180,E1 -20497.553,E2 -20497.553} C_VEL
LIN {X 0,Y 220.978,Z 556.946,A -85,B 0,C 180,E1 -20502.57,E2 -20502.57} C_VEL
LIN {X 0,Y 221.02,Z 556.954,A -85,B 0,C 180,E1 -20507.139,E2 -20507.139} C_VEL
LIN {X 0,Y 221.23,Z 556.909,A -85,B 0,C 180,E1 -20510.86,E2 -20510.86} C_VEL
LIN {X 0,Y 221.3,Z 556.917,A -85,B 0,C 180,E1 -20512.702,E2 -20512.702} C_VEL
LIN {X 0,Y 221.507,Z 556.879,A -85,B 0,C 180,E1 -20518.182,E2 -20518.182} C_VEL
LIN {X 0,Y 221.507,Z 556.885,A -85,B 0,C 180,E1 -20521.818,E2 -20521.818} C_VEL
LIN {X 0,Y 221.305,Z 556.919,A -85,B 0,C 180,E1 -20527.298,E2 -20527.298} C_VEL
LIN {X 0,Y 221.111,Z 556.927,A -85,B 0,C 180,E1 -20530.994,E2 -20530.994} C_VEL
LIN {X 0,Y 220.981,Z 556.95,A -85,B 0,C 180,E1 -20534.52,E2 -20534.52} C_VEL
LIN {X 0,Y 220.683,Z 556.99,A -85,B 0,C 180,E1 -20535.537,E2 -20535.537} C_VEL
LIN {X 0,Y 219.315,Z 557.165,A -85,B 0,C 180,E1 -20537.037,E2 -20537.037} C_VEL
LIN {X 0,Y 214.899,Z 557.708,A -85,B 0,C 180,E1 -20540.542,E2 -20540.542} C_VEL
LIN {X 0,Y 213.877,Z 557.831,A -85,B 0,C 180,E1 -20542.118,E2 -20542.118} C_VEL
LIN {X 0,Y 213.819,Z 557.841,A -85,B 0,C 180,E1 -20542.652,E2 -20542.652} C_VEL
LIN {X 0,Y 213.823,Z 557.841,A -85,B 0,C 180,E1 -20547.451,E2 -20547.451} C_VEL
LIN {X 0,Y 213.762,Z 557.851,A -85,B 0,C 180,E1 -20551.739,E2 -20551.739} C_VEL
LIN {X 0,Y 213.738,Z 557.829,A -85,B 0,C 180,E1 -20556.289,E2 -20556.289} C_VEL
LIN {X 0,Y 213.75,Z 557.848,A -85,B 0,C 180,E1 -20560.87,E2 -20560.87} C_VEL
LIN {X 0,Y 213.809,Z 557.914,A -85,B 0,C 180,E1 -20565.806,E2 -20565.806} C_VEL
LIN {X 0,Y 215.704,Z 565.1,A -85,B 0,C 180,E1 -20570.011,E2 -20570.011} C_VEL
LIN {X 0,Y 216.135,Z 566.479,A -85,B 0,C 180,E1 -20570.581,E2 -20570.581} C_VEL
LIN {X 0,Y 223.238,Z 580.132,A -85,B 0,C 180,E1 -20572.647,E2 -20572.647} C_VEL
LIN {X 0,Y 230.842,Z 596.806,A -85,B 0,C 180,E1 -20574.689,E2 -20574.689} C_VEL
LIN {X 0,Y 234.061,Z 604.875,A -85,B 0,C 180,E1 -20575.535,E2 -20575.535} C_VEL
LIN {X 0,Y 236.298,Z 621.283,A -85,B 0,C 180,E1 -20576.491,E2 -20576.491} C_VEL
LIN {X 0,Y 234.048,Z 675.098,A -85,B 0,C 180,E1 -20578.105,E2 -20578.105} C_VEL
LIN {X 0,Y 232.7,Z 688.486,A -85,B 0,C 180,E1 -20578.808,E2 -20578.808} C_VEL
LIN {X 0,Y 230.912,Z 700.392,A -85,B 0,C 180,E1 -20579.731,E2 -20579.731} C_VEL
LIN {X 0,Y 228.661,Z 712.6,A -85,B 0,C 180,E1 -20581.05,E2 -20581.05} C_VEL
LIN {X 0,Y 226.059,Z 724.162,A -85,B 0,C 180,E1 -20582.707,E2 -20582.707} C_VEL
LIN {X 0,Y 223.403,Z 734.576,A -85,B 0,C 180,E1 -20584.621,E2 -20584.621} C_VEL
LIN {X 0,Y 221.02,Z 743.095,A -85,B 0,C 180,E1 -20586.581,E2 -20586.581} C_VEL
LIN {X 0,Y 218.405,Z 752.334,A -85,B 0,C 180,E1 -20589.272,E2 -20589.272} C_VEL
LIN {X 0,Y 216.108,Z 759.762,A -85,B 0,C 180,E1 -20592.006,E2 -20592.006} C_VEL
LIN {X 0,Y 214.21,Z 765.726,A -85,B 0,C 180,E1 -20594.785,E2 -20594.785} C_VEL
LIN {X 0,Y 212.909,Z 770.445,A -85,B 0,C 180,E1 -20597.612,E2 -20597.612} C_VEL
LIN {X 0,Y 212.064,Z 774.059,A -85,B 0,C 180,E1 -20600.464,E2 -20600.464} C_VEL
LIN {X 0,Y 211.687,Z 775.921,A -85,B 0,C 180,E1 -20602.37,E2 -20602.37} C_VEL
LIN {X 0,Y 211.393,Z 778.174,A -85,B 0,C 180,E1 -20605.857,E2 -20605.857} C_VEL
LIN {X 0,Y 211.424,Z 778.926,A -85,B 0,C 180,E1 -20608.097,E2 -20608.097} C_VEL
LIN {X 0,Y 211.521,Z 779.14,A -85,B 0,C 180,E1 -20610.002,E2 -20610.002} C_VEL
LIN {X 0,Y 211.722,Z 778.523,A -85,B 0,C 180,E1 -20613.57,E2 -20613.57} C_VEL
LIN {X 0,Y 211.762,Z 780.567,A -85,B 0,C 180,E1 -20615.716,E2 -20615.716} C_VEL
LIN {X 0,Y 212.005,Z 781.957,A -85,B 0,C 180,E1 -20617.621,E2 -20617.621} C_VEL
LIN {X 0,Y 212.462,Z 782.858,A -85,B 0,C 180,E1 -20619.522,E2 -20619.522} C_VEL
LIN {X 0,Y 213.256,Z 783.195,A -85,B 0,C 180,E1 -20621.406,E2 -20621.406} C_VEL
LIN {X 0,Y 214.274,Z 783.084,A -85,B 0,C 180,E1 -20623.275,E2 -20623.275} C_VEL
LIN {X 0,Y 215.507,Z 782.559,A -85,B 0,C 180,E1 -20625.125,E2 -20625.125} C_VEL
LIN {X 0,Y 217.021,Z 781.546,A -85,B 0,C 180,E1 -20626.947,E2 -20626.947} C_VEL
LIN {X 0,Y 219.834,Z 779.072,A -85,B 0,C 180,E1 -20629.615,E2 -20629.615} C_VEL
LIN {X 0,Y 223.242,Z 775.396,A -85,B 0,C 180,E1 -20632.198,E2 -20632.198} C_VEL
LIN {X 0,Y 227.126,Z 770.496,A -85,B 0,C 180,E1 -20634.693,E2 -20634.693} C_VEL
LIN {X 0,Y 231.54,Z 764.258,A -85,B 0,C 180,E1 -20637.086,E2 -20637.086} C_VEL
LIN {X 0,Y 236.44,Z 756.25,A -85,B 0,C 180,E1 -20639.372,E2 -20639.372} C_VEL
LIN {X 0,Y 240.9,Z 747.986,A -85,B 0,C 180,E1 -20641.189,E2 -20641.189} C_VEL
LIN {X 0,Y 246.196,Z 736.617,A -85,B 0,C 180,E1 -20643.091,E2 -20643.091} C_VEL
LIN {X 0,Y 249.763,Z 727.591,A -85,B 0,C 180,E1 -20644.249,E2 -20644.249} C_VEL
LIN {X 0,Y 253.51,Z 716.356,A -85,B 0,C 180,E1 -20645.361,E2 -20645.361} C_VEL
LIN {X 0,Y 256.583,Z 704.441,A -85,B 0,C 180,E1 -20646.263,E2 -20646.263} C_VEL
LIN {X 0,Y 265.7,Z 660.649,A -85,B 0,C 180,E1 -20648.563,E2 -20648.563} C_VEL
LIN {X 0,Y 269.426,Z 643.205,A -85,B 0,C 180,E1 -20649.432,E2 -20649.432} C_VEL
LIN {X 0,Y 267.883,Z 641.929,A -85,B 0,C 180,E1 -20651.776,E2 -20651.776} C_VEL
LIN {X 0,Y 266.952,Z 642.02,A -85,B 0,C 180,E1 -20654.277,E2 -20654.277} C_VEL
LIN {X 0,Y 266.781,Z 643.571,A -85,B 0,C 180,E1 -20656.672,E2 -20656.672} C_VEL
LIN {X 0,Y 266.945,Z 645.155,A -85,B 0,C 180,E1 -20658.06,E2 -20658.06} C_VEL
LIN {X 0,Y 267.452,Z 649.017,A -85,B 0,C 180,E1 -20660.124,E2 -20660.124} C_VEL
LIN {X 0,Y 266.587,Z 660.167,A -85,B 0,C 180,E1 -20662.022,E2 -20662.022} C_VEL
LIN {X 0,Y 265.978,Z 668.759,A -85,B 0,C 180,E1 -20663.239,E2 -20663.239} C_VEL
LIN {X 0,Y 258.709,Z 704.898,A -85,B 0,C 180,E1 -20665.087,E2 -20665.087} C_VEL
LIN {X 0,Y 255.52,Z 716.646,A -85,B 0,C 180,E1 -20665.914,E2 -20665.914} C_VEL
LIN {X 0,Y 252.13,Z 726.391,A -85,B 0,C 180,E1 -20666.837,E2 -20666.837} C_VEL
LIN {X 0,Y 247.414,Z 737.891,A -85,B 0,C 180,E1 -20668.297,E2 -20668.297} C_VEL
LIN {X 0,Y 243.402,Z 746.115,A -85,B 0,C 180,E1 -20669.649,E2 -20669.649} C_VEL
LIN {X 0,Y 238.709,Z 754.499,A -85,B 0,C 180,E1 -20671.417,E2 -20671.417} C_VEL
LIN {X 0,Y 233.511,Z 762.588,A -85,B 0,C 180,E1 -20673.645,E2 -20673.645} C_VEL
LIN {X 0,Y 229.563,Z 767.888,A -85,B 0,C 180,E1 -20675.588,E2 -20675.588} C_VEL
LIN {X 0,Y 225.332,Z 772.851,A -85,B 0,C 180,E1 -20678.021,E2 -20678.021} C_VEL
LIN {X 0,Y 221.689,Z 776.57,A -85,B 0,C 180,E1 -20680.557,E2 -20680.557} C_VEL
LIN {X 0,Y 218.484,Z 779.086,A -85,B 0,C 180,E1 -20683.172,E2 -20683.172} C_VEL
LIN {X 0,Y 216.751,Z 780.062,A -85,B 0,C 180,E1 -20684.966,E2 -20684.966} C_VEL
LIN {X 0,Y 215.248,Z 780.578,A -85,B 0,C 180,E1 -20686.788,E2 -20686.788} C_VEL
LIN {X 0,Y 214.069,Z 780.653,A -85,B 0,C 180,E1 -20688.639,E2 -20688.639} C_VEL
LIN {X 0,Y 213.156,Z 780.266,A -85,B 0,C 180,E1 -20690.511,E2 -20690.511} C_VEL
LIN {X 0,Y 212.136,Z 778.387,A -85,B 0,C 180,E1 -20693.673,E2 -20693.673} C_VEL
LIN {X 0,Y 211.736,Z 774.768,A -85,B 0,C 180,E1 -20697.146,E2 -20697.146} C_VEL
LIN {X 0,Y 211.773,Z 770.421,A -85,B 0,C 180,E1 -20700,E2 -20700} C_VEL
LIN {X 0,Y 212.057,Z 764.37,A -85,B 0,C 180,E1 -20702.85,E2 -20702.85} C_VEL
LIN {X 0,Y 212.306,Z 757.94,A -85,B 0,C 180,E1 -20705.223,E2 -20705.223} C_VEL
LIN {X 0,Y 212.662,Z 749.939,A -85,B 0,C 180,E1 -20707.596,E2 -20707.596} C_VEL
LIN {X 0,Y 213.183,Z 740.764,A -85,B 0,C 180,E1 -20709.727,E2 -20709.727} C_VEL
LIN {X 0,Y 213.813,Z 730.694,A -85,B 0,C 180,E1 -20711.615,E2 -20711.615} C_VEL
LIN {X 0,Y 214.513,Z 719.079,A -85,B 0,C 180,E1 -20713.258,E2 -20713.258} C_VEL
LIN {X 0,Y 215.011,Z 708.14,A -85,B 0,C 180,E1 -20714.432,E2 -20714.432} C_VEL
LIN {X 0,Y 215.399,Z 694.796,A -85,B 0,C 180,E1 -20715.434,E2 -20715.434} C_VEL
LIN {X 0,Y 216.845,Z 644.931,A -85,B 0,C 180,E1 -20718.299,E2 -20718.299} C_VEL
LIN {X 0,Y 215.207,Z 622.636,A -85,B 0,C 180,E1 -20719.585,E2 -20719.585} C_VEL
LIN {X 0,Y 215.177,Z 617.284,A -85,B 0,C 180,E1 -20719.957,E2 -20719.957} C_VEL
LIN {X 0,Y 217.145,Z 596.54,A -85,B 0,C 180,E1 -20725.343,E2 -20725.343} C_VEL
LIN {X 0,Y 218.723,Z 581.989,A -85,B 0,C 180,E1 -20729.107,E2 -20729.107} C_VEL
LIN {X 0,Y 215.745,Z 566.867,A -85,B 0,C 180,E1 -20733.277,E2 -20733.277} C_VEL
LIN {X 0,Y 213.916,Z 557.997,A -85,B 0,C 180,E1 -20735.857,E2 -20735.857} C_VEL
LIN {X 0,Y 213.718,Z 557.799,A -85,B 0,C 180,E1 -20741.124,E2 -20741.124} C_VEL
LIN {X 0,Y 213.708,Z 557.804,A -85,B 0,C 180,E1 -20743.679,E2 -20743.679} C_VEL
LIN {X 0,Y 213.709,Z 557.863,A -85,B 0,C 180,E1 -20746.344,E2 -20746.344} C_VEL
LIN {X 0,Y 213.79,Z 558.069,A -85,B 0,C 180,E1 -20750.012,E2 -20750.012} C_VEL
LIN {X 0,Y 214.066,Z 559.156,A -85,B 0,C 180,E1 -20750.37,E2 -20750.37} C_VEL
LIN {X 0,Y 215.536,Z 561.731,A -85,B 0,C 180,E1 -20750.825,E2 -20750.825} C_VEL
LIN {X 0,Y 216.647,Z 563.25,A -85,B 0,C 180,E1 -20751.129,E2 -20751.129} C_VEL
LIN {X 0,Y 222.79,Z 573.228,A -85,B 0,C 180,E1 -20752.8,E2 -20752.8} C_VEL
LIN {X 0,Y 230.498,Z 588.786,A -85,B 0,C 180,E1 -20754.836,E2 -20754.836} C_VEL
LIN {X 0,Y 235.816,Z 601.446,A -85,B 0,C 180,E1 -20756.206,E2 -20756.206} C_VEL
LIN {X 0,Y 236.936,Z 604.941,A -85,B 0,C 180,E1 -20756.514,E2 -20756.514} C_VEL
LIN {X 0,Y 234.333,Z 664.172,A -85,B 0,C 180,E1 -20758.275,E2 -20758.275} C_VEL
LIN {X 0,Y 233.08,Z 677.481,A -85,B 0,C 180,E1 -20759.001,E2 -20759.001} C_VEL
LIN {X 0,Y 231.351,Z 690.193,A -85,B 0,C 180,E1 -20760.042,E2 -20760.042} C_VEL
LIN {X 0,Y 229.265,Z 701.982,A -85,B 0,C 180,E1 -20761.38,E2 -20761.38} C_VEL
LIN {X 0,Y 226.796,Z 713.32,A -85,B 0,C 180,E1 -20763.049,E2 -20763.049} C_VEL
LIN {X 0,Y 224.268,Z 723.535,A -85,B 0,C 180,E1 -20764.971,E2 -20764.971} C_VEL
LIN {X 0,Y 221.736,Z 733.208,A -85,B 0,C 180,E1 -20767.308,E2 -20767.308} C_VEL
LIN {X 0,Y 219.156,Z 741.6,A -85,B 0,C 180,E1 -20769.833,E2 -20769.833} C_VEL
LIN {X 0,Y 216.863,Z 748.765,A -85,B 0,C 180,E1 -20772.555,E2 -20772.555} C_VEL
LIN {X 0,Y 215.316,Z 753.596,A -85,B 0,C 180,E1 -20774.862,E2 -20774.862} C_VEL
LIN {X 0,Y 213.779,Z 758.289,A -85,B 0,C 180,E1 -20777.66,E2 -20777.66} C_VEL
LIN {X 0,Y 212.74,Z 761.871,A -85,B 0,C 180,E1 -20780.491,E2 -20780.491} C_VEL
LIN {X 0,Y 212.244,Z 763.722,A -85,B 0,C 180,E1 -20782.387,E2 -20782.387} C_VEL
LIN {X 0,Y 211.893,Z 765.113,A -85,B 0,C 180,E1 -20784.288,E2 -20784.288} C_VEL
LIN {X 0,Y 211.694,Z 766.103,A -85,B 0,C 180,E1 -20786.191,E2 -20786.191} C_VEL
LIN {X 0,Y 211.596,Z 766.711,A -85,B 0,C 180,E1 -20788.095,E2 -20788.095} C_VEL
LIN {X 0,Y 211.58,Z 766.939,A -85,B 0,C 180,E1 -20789.998,E2 -20789.998} C_VEL
LIN {X 0,Y 211.595,Z 766.747,A -85,B 0,C 180,E1 -20791.902,E2 -20791.902} C_VEL
LIN {X 0,Y 211.692,Z 766.163,A -85,B 0,C 180,E1 -20793.805,E2 -20793.805} C_VEL
LIN {X 0,Y 212.242,Z 763.842,A -85,B 0,C 180,E1 -20797.61,E2 -20797.61} C_VEL
LIN {X 0,Y 213.016,Z 760.973,A -85,B 0,C 180,E1 -20800.453,E2 -20800.453} C_VEL
LIN {X 0,Y 214.206,Z 757.08,A -85,B 0,C 180,E1 -20803.276,E2 -20803.276} C_VEL
LIN {X 0,Y 215.862,Z 752.06,A -85,B 0,C 180,E1 -20806.064,E2 -20806.064} C_VEL
LIN {X 0,Y 217.856,Z 745.737,A -85,B 0,C 180,E1 -20808.818,E2 -20808.818} C_VEL
LIN {X 0,Y 220.444,Z 737.817,A -85,B 0,C 180,E1 -20811.506,E2 -20811.506} C_VEL
LIN {X 0,Y 222.833,Z 729.264,A -85,B 0,C 180,E1 -20813.844,E2 -20813.844} C_VEL
LIN {X 0,Y 225.24,Z 719.9,A -85,B 0,C 180,E1 -20815.9,E2 -20815.9} C_VEL
LIN {X 0,Y 227.876,Z 708.808,A -85,B 0,C 180,E1 -20817.804,E2 -20817.804} C_VEL
LIN {X 0,Y 230.197,Z 697.923,A -85,B 0,C 180,E1 -20819.239,E2 -20819.239} C_VEL
LIN {X 0,Y 232.122,Z 685.888,A -85,B 0,C 180,E1 -20820.472,E2 -20820.472} C_VEL
LIN {X 0,Y 233.607,Z 673.45,A -85,B 0,C 180,E1 -20821.39,E2 -20821.39} C_VEL
LIN {X 0,Y 234.686,Z 660.698,A -85,B 0,C 180,E1 -20821.979,E2 -20821.979} C_VEL
LIN {X 0,Y 236.969,Z 604.266,A -85,B 0,C 180,E1 -20823.648,E2 -20823.648} C_VEL
LIN {X 0,Y 231.162,Z 590.237,A -85,B 0,C 180,E1 -20825.14,E2 -20825.14} C_VEL
LIN {X 0,Y 223.048,Z 573.631,A -85,B 0,C 180,E1 -20827.288,E2 -20827.288} C_VEL
LIN {X 0,Y 217.941,Z 565.424,A -85,B 0,C 180,E1 -20828.663,E2 -20828.663} C_VEL
LIN {X 0,Y 216.004,Z 562.204,A -85,B 0,C 180,E1 -20829.213,E2 -20829.213} C_VEL
LIN {X 0,Y 214.284,Z 559.762,A -85,B 0,C 180,E1 -20829.697,E2 -20829.697} C_VEL
LIN {X 0,Y 213.763,Z 557.841,A -85,B 0,C 180,E1 -20829.951,E2 -20829.951} C_VEL
LIN {X 0,Y 213.705,Z 557.847,A -85,B 0,C 180,E1 -20833.676,E2 -20833.676} C_VEL
LIN {X 0,Y 213.744,Z 557.843,A -85,B 0,C 180,E1 -20836.331,E2 -20836.331} C_VEL
LIN {X 0,Y 213.758,Z 557.844,A -85,B 0,C 180,E1 -20839.127,E2 -20839.127} C_VEL
LIN {X 0,Y 213.749,Z 557.845,A -85,B 0,C 180,E1 -20843.713,E2 -20843.713} C_VEL
LIN {X 0,Y 213.791,Z 557.849,A -85,B 0,C 180,E1 -20848.723,E2 -20848.723} C_VEL
LIN {X 0,Y 213.821,Z 557.836,A -85,B 0,C 180,E1 -20852.602,E2 -20852.602} C_VEL
LIN {X 0,Y 213.846,Z 557.834,A -85,B 0,C 180,E1 -20856.952,E2 -20856.952} C_VEL
LIN {X 0,Y 213.926,Z 557.827,A -85,B 0,C 180,E1 -20862.304,E2 -20862.304} C_VEL
LIN {X 0,Y 213.974,Z 557.83,A -85,B 0,C 180,E1 -20866.708,E2 -20866.708} C_VEL
LIN {X 0,Y 214.161,Z 557.788,A -85,B 0,C 180,E1 -20870.556,E2 -20870.556} C_VEL
LIN {X 0,Y 214.234,Z 557.796,A -85,B 0,C 180,E1 -20872.46,E2 -20872.46} C_VEL
LIN {X 0,Y 214.44,Z 557.758,A -85,B 0,C 180,E1 -20878.122,E2 -20878.122} C_VEL
LIN {X 0,Y 214.548,Z 557.761,A -85,B 0,C 180,E1 -20880,E2 -20880} C_VEL
LIN {X 0,Y 214.44,Z 557.765,A -85,B 0,C 180,E1 -20881.878,E2 -20881.878} C_VEL
LIN {X 0,Y 214.242,Z 557.797,A -85,B 0,C 180,E1 -20887.54,E2 -20887.54} C_VEL
LIN {X 0,Y 214.041,Z 557.81,A -85,B 0,C 180,E1 -20891.362,E2 -20891.362} C_VEL
LIN {X 0,Y 213.927,Z 557.824,A -85,B 0,C 180,E1 -20895.237,E2 -20895.237} C_VEL
LIN {X 0,Y 213.862,Z 557.846,A -85,B 0,C 180,E1 -20899.185,E2 -20899.185} C_VEL
LIN {X 0,Y 213.819,Z 557.841,A -85,B 0,C 180,E1 -20902.652,E2 -20902.652} C_VEL
LIN {X 0,Y 213.549,Z 557.883,A -85,B 0,C 180,E1 -20903.704,E2 -20903.704} C_VEL
LIN {X 0,Y 212.224,Z 558.051,A -85,B 0,C 180,E1 -20905.258,E2 -20905.258} C_VEL
LIN {X 0,Y 207.845,Z 558.596,A -85,B 0,C 180,E1 -20908.889,E2 -20908.889} C_VEL
LIN {X 0,Y 206.779,Z 558.72,A -85,B 0,C 180,E1 -20910.522,E2 -20910.522} C_VEL
LIN {X 0,Y 206.695,Z 558.729,A -85,B 0,C 180,E1 -20911.075,E2 -20911.075} C_VEL
LIN {X 0,Y 206.694,Z 558.712,A -85,B 0,C 180,E1 -20915.312,E2 -20915.312} C_VEL
LIN {X 0,Y 206.746,Z 558.716,A -85,B 0,C 180,E1 -20918.573,E2 -20918.573} C_VEL
LIN {X 0,Y 206.674,Z 558.719,A -85,B 0,C 180,E1 -20922.852,E2 -20922.852} C_VEL
LIN {X 0,Y 206.751,Z 558.922,A -85,B 0,C 180,E1 -20924.673,E2 -20924.673} C_VEL
LIN {X 0,Y 208.62,Z 565.807,A -85,B 0,C 180,E1 -20928.781,E2 -20928.781} C_VEL
LIN {X 0,Y 210.856,Z 570.096,A -85,B 0,C 180,E1 -20929.613,E2 -20929.613} C_VEL
LIN {X 0,Y 216.306,Z 580.125,A -85,B 0,C 180,E1 -20931.241,E2 -20931.241} C_VEL
LIN {X 0,Y 223.162,Z 594.656,A -85,B 0,C 180,E1 -20933.205,E2 -20933.205} C_VEL
LIN {X 0,Y 228.43,Z 607.684,A -85,B 0,C 180,E1 -20934.672,E2 -20934.672} C_VEL
LIN {X 0,Y 230.388,Z 622.833,A -85,B 0,C 180,E1 -20935.576,E2 -20935.576} C_VEL
LIN {X 0,Y 228.061,Z 674.686,A -85,B 0,C 180,E1 -20937.151,E2 -20937.151} C_VEL
LIN {X 0,Y 226.75,Z 687.729,A -85,B 0,C 180,E1 -20937.845,E2 -20937.845} C_VEL
LIN {X 0,Y 224.808,Z 700.194,A -85,B 0,C 180,E1 -20938.819,E2 -20938.819} C_VEL
LIN {X 0,Y 222.478,Z 712.4,A -85,B 0,C 180,E1 -20940.165,E2 -20940.165} C_VEL
LIN {X 0,Y 219.761,Z 723.961,A -85,B 0,C 180,E1 -20941.857,E2 -20941.857} C_VEL
LIN {X 0,Y 216.977,Z 734.373,A -85,B 0,C 180,E1 -20943.814,E2 -20943.814} C_VEL
LIN {X 0,Y 214.488,Z 742.892,A -85,B 0,C 180,E1 -20945.823,E2 -20945.823} C_VEL
LIN {X 0,Y 212.335,Z 750.16,A -85,B 0,C 180,E1 -20947.936,E2 -20947.936} C_VEL
LIN {X 0,Y 210.049,Z 757.28,A -85,B 0,C 180,E1 -20950.454,E2 -20950.454} C_VEL
LIN {X 0,Y 207.956,Z 763.701,A -85,B 0,C 180,E1 -20953.308,E2 -20953.308} C_VEL
LIN {X 0,Y 206.322,Z 768.804,A -85,B 0,C 180,E1 -20956.207,E2 -20956.207} C_VEL
LIN {X 0,Y 205.29,Z 772.778,A -85,B 0,C 180,E1 -20959.149,E2 -20959.149} C_VEL
LIN {X 0,Y 204.639,Z 775.716,A -85,B 0,C 180,E1 -20962.106,E2 -20962.106} C_VEL
LIN {X 0,Y 204.401,Z 777.113,A -85,B 0,C 180,E1 -20964.081,E2 -20964.081} C_VEL
LIN {X 0,Y 204.329,Z 778.721,A -85,B 0,C 180,E1 -20968.031,E2 -20968.031} C_VEL
LIN {X 0,Y 204.421,Z 778.935,A -85,B 0,C 180,E1 -20970.002,E2 -20970.002} C_VEL
LIN {X 0,Y 204.666,Z 778.125,A -85,B 0,C 180,E1 -20973.94,E2 -20973.94} C_VEL
LIN {X 0,Y 204.699,Z 778.124,A -85,B 0,C 180,E1 -20974.274,E2 -20974.274} C_VEL
LIN {X 0,Y 205.005,Z 781.356,A -85,B 0,C 180,E1 -20977.883,E2 -20977.883} C_VEL
LIN {X 0,Y 205.468,Z 782.373,A -85,B 0,C 180,E1 -20979.849,E2 -20979.849} C_VEL
LIN {X 0,Y 206.289,Z 782.979,A -85,B 0,C 180,E1 -20981.797,E2 -20981.797} C_VEL
LIN {X 0,Y 207.377,Z 783.169,A -85,B 0,C 180,E1 -20983.725,E2 -20983.725} C_VEL
LIN {X 0,Y 208.673,Z 782.814,A -85,B 0,C 180,E1 -20985.632,E2 -20985.632} C_VEL
LIN {X 0,Y 210.266,Z 781.976,A -85,B 0,C 180,E1 -20987.508,E2 -20987.508} C_VEL
LIN {X 0,Y 212.104,Z 780.725,A -85,B 0,C 180,E1 -20989.352,E2 -20989.352} C_VEL
LIN {X 0,Y 215.568,Z 777.868,A -85,B 0,C 180,E1 -20992.021,E2 -20992.021} C_VEL
LIN {X 0,Y 219.506,Z 773.909,A -85,B 0,C 180,E1 -20994.598,E2 -20994.598} C_VEL
LIN {X 0,Y 223.943,Z 768.692,A -85,B 0,C 180,E1 -20997.07,E2 -20997.07} C_VEL
LIN {X 0,Y 228.873,Z 761.965,A -85,B 0,C 180,E1 -20999.428,E2 -20999.428} C_VEL
LIN {X 0,Y 233.402,Z 754.972,A -85,B 0,C 180,E1 -21001.295,E2 -21001.295} C_VEL
LIN {X 0,Y 237.27,Z 748.404,A -85,B 0,C 180,E1 -21002.724,E2 -21002.724} C_VEL
LIN {X 0,Y 242.404,Z 738.437,A -85,B 0,C 180,E1 -21004.429,E2 -21004.429} C_VEL
LIN {X 0,Y 246.743,Z 728.451,A -85,B 0,C 180,E1 -21005.727,E2 -21005.727} C_VEL
LIN {X 0,Y 250.136,Z 719.312,A -85,B 0,C 180,E1 -21006.661,E2 -21006.661} C_VEL
LIN {X 0,Y 253.825,Z 706.783,A -85,B 0,C 180,E1 -21007.654,E2 -21007.654} C_VEL
LIN {X 0,Y 258.83,Z 684.465,A -85,B 0,C 180,E1 -21008.908,E2 -21008.908} C_VEL
LIN {X 0,Y 266.729,Z 649.274,A -85,B 0,C 180,E1 -21010.633,E2 -21010.633} C_VEL
LIN {X 0,Y 265.818,Z 648.737,A -85,B 0,C 180,E1 -21012.243,E2 -21012.243} C_VEL
LIN {X 0,Y 265.095,Z 649.079,A -85,B 0,C 180,E1 -21014.712,E2 -21014.712} C_VEL
LIN {X 0,Y 265.02,Z 651.138,A -85,B 0,C 180,E1 -21017.257,E2 -21017.257} C_VEL
LIN {X 0,Y 265.254,Z 654.632,A -85,B 0,C 180,E1 -21019.242,E2 -21019.242} C_VEL
LIN {X 0,Y 264.016,Z 665.64,A -85,B 0,C 180,E1 -21021.093,E2 -21021.093} C_VEL
LIN {X 0,Y 263.399,Z 671.361,A -85,B 0,C 180,E1 -21021.89,E2 -21021.89} C_VEL
LIN {X 0,Y 256.456,Z 704.008,A -85,B 0,C 180,E1 -21023.535,E2 -21023.535} C_VEL
LIN {X 0,Y 253.125,Z 715.828,A -85,B 0,C 180,E1 -21024.334,E2 -21024.334} C_VEL
LIN {X 0,Y 248.949,Z 727.044,A -85,B 0,C 180,E1 -21025.379,E2 -21025.379} C_VEL
LIN {X 0,Y 243.981,Z 738.437,A -85,B 0,C 180,E1 -21026.818,E2 -21026.818} C_VEL
LIN {X 0,Y 239.734,Z 746.488,A -85,B 0,C 180,E1 -21028.151,E2 -21028.151} C_VEL
LIN {X 0,Y 234.686,Z 754.794,A -85,B 0,C 180,E1 -21029.894,E2 -21029.894} C_VEL
LIN {X 0,Y 229.177,Z 762.783,A -85,B 0,C 180,E1 -21032.117,E2 -21032.117} C_VEL
LIN {X 0,Y 224.905,Z 768.005,A -85,B 0,C 180,E1 -21034.057,E2 -21034.057} C_VEL
LIN {X 0,Y 220.324,Z 772.977,A -85,B 0,C 180,E1 -21036.501,E2 -21036.501} C_VEL
LIN {X 0,Y 216.298,Z 776.64,A -85,B 0,C 180,E1 -21039.058,E2 -21039.058} C_VEL
LIN {X 0,Y 213.947,Z 778.381,A -85,B 0,C 180,E1 -21040.823,E2 -21040.823} C_VEL
LIN {X 0,Y 211.723,Z 779.677,A -85,B 0,C 180,E1 -21042.618,E2 -21042.618} C_VEL
LIN {X 0,Y 209.922,Z 780.506,A -85,B 0,C 180,E1 -21044.465,E2 -21044.465} C_VEL
LIN {X 0,Y 208.357,Z 780.789,A -85,B 0,C 180,E1 -21046.343,E2 -21046.343} C_VEL
LIN {X 0,Y 207.11,Z 780.568,A -85,B 0,C 180,E1 -21048.252,E2 -21048.252} C_VEL
LIN {X 0,Y 206.174,Z 779.919,A -85,B 0,C 180,E1 -21050.187,E2 -21050.187} C_VEL
LIN {X 0,Y 205.491,Z 778.839,A -85,B 0,C 180,E1 -21052.137,E2 -21052.137} C_VEL
LIN {X 0,Y 204.82,Z 776.025,A -85,B 0,C 180,E1 -21055.2,E2 -21055.2} C_VEL
